   VAR_TEMP 
      tempExecute : Bool;
      tempNumberOfPoints : Int;
   END_VAR

   VAR CONSTANT 
      FB_STATE_NO_PROCESSING : DInt := 0;
      FB_STATE_ENABLE_MOVE_TO_END_POS : DInt := 3;
      FB_STATE_MOVE_TO_END_POSITION : DInt := 4;
      FB_STATE_ENABLE_RAMP_UP : DInt := 6;
      FB_STATE_RAMP_UP : DInt := 9;
      FB_STATE_WAIT_FOR_MEASUREMENT : DInt := 10;
      FB_STATE_MEASUREMENT : DInt := 11;
      FB_STATE_RAMP_DOWN : DInt := 12;
      FB_STATE_ERROR : DInt := 16;
      FB_STATE_COMMAND_ABORTED : DInt := 17;
      UNDEFINED : Byte;
      FORWARD : Byte := 16#1;
      BACKWARD : Byte := 16#2;
      FINE_RANGE : Int := 0;
      COARSE_RANGE : Int := 1;
      STATUS_MEASUREMENT_OK : Word := 16#0000;
      STATUS_MEASUREMENT_MOVE_TO_END_POS : Word := 16#0001;
      STATUS_MEASUREMENT_WAITING : Word := 16#0002;
      STATUS_MEASUREMENT_BUSY : Word := 16#0004;
      STATUS_MEASUREMENT_IS_ABORTED : Word := 16#0008;
      STATUS_MEASUREMENT_DISTANCE_TO_SMALL : Word := 16#0010;
      STATUS_MEASUREMENT_ARRAY_FORWARD_LIMITED : Word := 16#0020;
      STATUS_MEASUREMENT_ARRAY_BACKWARD_LIMITED : Word := 16#0040;
      STATUS_MEASUREMENT_ERROR : Word := 16#8000;
      STATUS_EXECUTION_FINISHED : Word := 16#0000;
      STATUS_NO_CALL : Word := 16#7000;
      STATUS_FIRST_CALL : Word := 16#7001;
      STATUS_SUBSEQUENT_CALL : Word := 16#7002;
      STATUS_WAITING_FOR_ENABLING_FORWARD : Word := 16#7003;
      STATUS_WAITING_FOR_ENABLING_BACKWARD : Word := 16#7004;
      ALARM_MEASUREMENT_IS_RUNNING : Word := 16#8201;
      ALARM_ABORT_IS_ON : Word := 16#8202;
      ALARM_UNDEFINED_STATE : Word := 16#8600;
      ALARM_VALUE_RAMP_FORWARTS : Word := 16#8005;
      ALARM_VALUE_RAMP_BACKWARDS : Word := 16#8006;
      ALARM_DIRECTION : Word := 16#8007;
      ALARM_VALUE_TRAVERSING_DISTANCE : Word := 16#8010;
      ALARM_VALUE_MAX_VELOCITY : Word := 16#8011;
      ALARM_CONFIGURATION : Word := 16#8012;
      ALARM_AXIS_ERROR_OCCURED : Word := 16#8001;
      ALARM_AXIS_DISABLED : Word := 16#800F;
   END_VAR


BEGIN
	//================================================================================
	//SIEMENS AG // (c)Copyright 2019 All Rights Reserved
	//--------------------------------------------------------------------------------
	//Library:       LSimaHydTO
	//Tested with:   S7-15xx
	//Engineering:   TIA Portal  V15
	//Restrictions:  -
	//Requirements:  S7-1500 (FW 2.5)
	//Functionality: Execute valve characteristic measurement
	//
	//--------------------------------------------------------------------------------
	//Change log table:
	//
	//Version     Date          Expert in charge    Changes applied
	//01.00    15.03.2018    APC_ERLF            First released version
	//01.22    22.04.2020    APC_ERLF              - improved: units are taken into account for the control
	//================================================================================
	#tempExecute := #execute; // Work with temporary value / create process image
	
	REGION TRIGGERING
	  IF #tempExecute AND NOT #statExecuteOld  // Check if FB is triggered
	  THEN // First call; initialize FB
	    IF #statStatus <> #STATUS_NO_CALL THEN
	      #statFBState := #FB_STATE_ERROR;
	      #statStatus := #ALARM_MEASUREMENT_IS_RUNNING;
	    ELSIF #abort THEN
	      #statFBState := #FB_STATE_ERROR;
	      #statStatus := #ALARM_ABORT_IS_ON;
	    ELSE
	      
	      #statDone := FALSE;
	      #statBusy := TRUE;
	      #statError := FALSE;
	      #statCommandAborted := FALSE;
	      #statStatus := #STATUS_FIRST_CALL;
	      
	      // reset outputs 
	      #qOutputValueStepBackward := 0.0;
	      #qOutputValueStepForward := 0.0;
	      #velocityStepBackward := 0.0;
	      #velocityStepForward := 0.0;
	      #statDirection := #UNDEFINED;
	      #statStatusMeasurement := #STATUS_MEASUREMENT_OK;
	      #statIdx := "LSIMAHYD_VCHAR_POINTS_UPPER_LIMIT" + 1;
	      
	      "LSimaHydTO_CheckPlausibilityConfigData"(forwardFineRangeStepValue => #statForwardFineRangeStepValue,
	                                               forwardCoarseRangeStepValue => #statForwardCoarseRangeStepValue,
	                                               backwardFineRangeStepValue => #statBackwardFineRangeStepValue,
	                                               backwardCoarseRangeStepValue => #statBackwardCoarseRangeStepValue,
	                                               configForwardOK => #statConfigForwardOK,
	                                               configBackwardOK => #statConfigBackwardOK,
	                                               configData := #configData);
	      
	      
	      REGION check input parameters
	        IF #axis.Internal.PositionLimits_SW.Active THEN
	          #statMaxPosition := #axis.Internal.PositionLimits_SW.MaxPosition - ABS(#configData.safetyDistance);
	          #statMinPosition := #axis.Internal.PositionLimits_SW.MinPosition + ABS(#configData.safetyDistance);
	          //check if actual position is in the limits
	        ELSE
	          #statMaxPosition := 1.0e12;
	          #statMinPosition := -1.0e12;
	          //check if actual position is in the limits
	        END_IF;
	        
	        IF #configData.forward.ramp = 0.0
	          AND #configData.forward.enableMeasurement
	        THEN
	          #statFBState := #FB_STATE_ERROR;
	          #statStatus := #ALARM_VALUE_RAMP_FORWARTS;
	        ELSIF #configData.backward.ramp = 0.0
	          AND #configData.backward.enableMeasurement
	        THEN
	          #statFBState := #FB_STATE_ERROR;
	          #statStatus := #ALARM_VALUE_RAMP_BACKWARDS;
	        ELSIF #statMaxPosition <= #statMinPosition
	          OR #configData.safetyDistance < 0.0
	        THEN
	          #statFBState := #FB_STATE_ERROR;
	          #statStatus := #ALARM_VALUE_TRAVERSING_DISTANCE;
	        ELSIF NOT (#configData.forward.enableMeasurement OR #configData.backward.enableMeasurement)
	        THEN
	          //error: no direction is enabled
	          #statFBState := #FB_STATE_ERROR;
	          #statStatus := #ALARM_DIRECTION;
	        ELSIF (#configData.forward.maxVelocity = 0.0 AND #configData.forward.enableMeasurement)
	          OR (#configData.backward.maxVelocity = 0.0 AND #configData.backward.enableMeasurement)
	        THEN
	          //error: illegal value Vmax
	          #statFBState := #FB_STATE_ERROR;
	          #statStatus := #ALARM_VALUE_MAX_VELOCITY;
	        ELSE
	          //check config forward
	          IF #statConfigForwardOK THEN
	            IF #configData.forward.fineRange.numberOfPoints > 0 THEN
	              #statRangeForward := #FINE_RANGE;
	              #statCoarseBeginForward := -1;
	            ELSE
	              #statRangeForward := #COARSE_RANGE;
	              #statCoarseBeginForward := 0;
	            END_IF;
	          END_IF;
	          //check config backward
	          IF #statConfigBackwardOK THEN
	            IF #configData.backward.fineRange.numberOfPoints > 0 THEN
	              #statRangeBackward := #FINE_RANGE;
	              #statCoarseBeginBackward := -1;
	            ELSE
	              #statRangeBackward := #COARSE_RANGE;
	              #statCoarseBeginBackward := 0;
	            END_IF;
	          END_IF;
	          IF NOT (#statConfigForwardOK OR #statConfigBackwardOK) THEN
	            //error: illegal config configuration
	            #statFBState := #FB_STATE_ERROR;
	            #statStatus := #ALARM_CONFIGURATION;
	          ELSE
	            #statError := FALSE;
	            #statStatus := #STATUS_FIRST_CALL;
	            #statStatusMeasurement := #STATUS_MEASUREMENT_OK;
	          END_IF;
	        END_IF;
	        
	        //check input parameters
	        IF #statFBState <> #FB_STATE_ERROR
	        THEN
	          //init internal variables
	          #statMeasurementForwardDone := NOT #configData.forward.enableMeasurement;
	          #statMeasurementBackwardDone := NOT #configData.backward.enableMeasurement;
	          #statActualStepForward := 0;
	          #statActualStepBackward := 0;
	          #statIdx := 0;
	          #measuredValues.forward.maxQOutput := 0.0;
	          #measuredValues.forward.maxVelocity := 0.0;
	          #measuredValues.forward.maxIndexMeasurement := -1;
	          #measuredValues.backward.maxQOutput := 0.0;
	          #measuredValues.backward.maxVelocity := 0.0;
	          #measuredValues.backward.maxIndexMeasurement := -1;
	          #statStepCounterMeasurementForwardAborted := 0;
	          #statStepCounterMeasurementBackwardAborted := 0;
	          
	        ELSE
	          //set PLCopen outputs
	          #statBusy := FALSE;
	        END_IF;
	        
	      END_REGION
	      
	    END_IF;
	  ELSIF (#statStatus = #STATUS_FIRST_CALL) THEN
	    #statStatus := #STATUS_SUBSEQUENT_CALL;
	  END_IF;
	  
	  // Edge detection 'execute' input
	  #statExecuteOld := #tempExecute;
	END_REGION TRIGGERING
	
	IF (#statStatus = #STATUS_NO_CALL) THEN // Nothing to do -> End here to reduce "system load"
	  RETURN;
	END_IF;
	
	REGION WATCHING 
	  //get actual position
	  #statActualPosition := #axis.ActualPosition;
	  //get actual Time
	  #statRetInt := RD_SYS_T(#statActualTime);
	  //init internal variables
	  
	  
	  REGION INIT_MEASUREMENT
	    IF #statStatus = #STATUS_FIRST_CALL AND NOT #statError THEN
	      #statStatusMeasurement := #statStatusMeasurement AND NOT #STATUS_MEASUREMENT_MOVE_TO_END_POS;
	      
	      IF #configData.forward.enableMeasurement AND #configData.backward.enableMeasurement THEN
	        //check start direction
	        IF (#statMaxPosition - #statActualPosition) > (#statActualPosition - #statMinPosition) THEN
	          #statDirection := #FORWARD;
	        ELSE
	          #statDirection := #BACKWARD;
	        END_IF;
	        #statFBState := #FB_STATE_ENABLE_RAMP_UP;
	      ELSE
	        IF #configData.forward.enableMeasurement THEN
	          IF #statActualPosition < #statMaxPosition - #configData.safetyDistance THEN
	            #statDirection := #FORWARD;
	            #statFBState := #FB_STATE_ENABLE_RAMP_UP;
	          ELSE
	            #statDirection := #BACKWARD;
	            #statFBState := #FB_STATE_ENABLE_MOVE_TO_END_POS;
	          END_IF;
	        ELSE
	          IF #statActualPosition > #statMinPosition + #configData.safetyDistance THEN
	            #statDirection := #BACKWARD;
	            #statFBState := #FB_STATE_ENABLE_RAMP_UP;
	          ELSE
	            #statDirection := #FORWARD;
	            #statFBState := #FB_STATE_ENABLE_MOVE_TO_END_POS;
	          END_IF;
	        END_IF;
	      END_IF;
	      //start always from min. value
	      #statQOutputForward := MAX(IN1 := #configData.forward.minQOutputValue, IN2 := #configData.offset);
	      #measuredValues.forward.minQOutput := (#configData.forward.minQOutputValue);
	      #statQOutputBackward := MAX(IN1 := ABS(#configData.backward.minQOutputValue), IN2 := ABS(#configData.offset));
	      #measuredValues.backward.minQOutput := (- #configData.backward.minQOutputValue);
	      #statEnableRamping := (#enableRampingForward AND #statDirection = #FORWARD) OR (#enableRampingBackward AND #statDirection = #BACKWARD);
	      
	    END_IF;
	  END_REGION INIT_MEASUREMENT
	  
	  
	  #statEnableRamping := (#enableRampingForward AND #statDirection = #FORWARD) OR (#enableRampingBackward AND #statDirection = #BACKWARD);
	  IF ((#axis.ErrorWord <> 0 OR NOT #axis.StatusActor.Enabled)
	    AND #statFBState <> #FB_STATE_NO_PROCESSING) OR  #statFBState = #FB_STATE_ERROR
	  THEN
	    IF #axis.ErrorWord <> 0 THEN
	      #statStatus := #ALARM_AXIS_ERROR_OCCURED;
	    ELSIF NOT #axis.StatusActor.Enabled THEN
	      #statStatus := #ALARM_AXIS_DISABLED;
	    END_IF;
	    
	    #axis.Internal.Control.DirectOutput.activate := FALSE;
	    #axis.Internal.Control.DirectOutput.jogForward := FALSE;
	    #axis.Internal.Control.DirectOutput.jogBackward := FALSE;
	    #statFBState := #FB_STATE_ERROR;
	    // stop/pause measurement
	  ELSIF (#abort AND NOT #statAbortOld)
	    OR
	    (NOT #statEnableRamping AND #statEnableRampingOld)
	  THEN
	    IF #statFBState = #FB_STATE_MOVE_TO_END_POSITION
	      OR #statFBState = #FB_STATE_RAMP_UP
	      OR #statFBState = #FB_STATE_WAIT_FOR_MEASUREMENT
	      OR #statFBState = #FB_STATE_MEASUREMENT THEN
	      #statCommandAborted := #abort;
	      #axis.Internal.Control.DirectOutput.jogForward := FALSE;
	      #axis.Internal.Control.DirectOutput.jogBackward := FALSE;
	      #statFBState := #FB_STATE_RAMP_DOWN;
	    ELSIF #abort AND #statFBState <> #FB_STATE_NO_PROCESSING
	      AND #statFBState <> #FB_STATE_ERROR
	      AND #statFBState <> #FB_STATE_COMMAND_ABORTED
	    THEN
	      #statCommandAborted := #abort;
	      #statStatusMeasurement := #STATUS_MEASUREMENT_IS_ABORTED;
	      #statFBState := #FB_STATE_COMMAND_ABORTED;
	    END_IF;
	  END_IF;
	  
	  
	  // do not use statI in a following operation
	  IF #statIdx <= "LSIMAHYD_VCHAR_POINTS_UPPER_LIMIT" THEN
	    #measuredValues.forward.qOutput[#statIdx] := 0.0;  // Q-Output value
	    #measuredValues.forward.velocity[#statIdx] := 0.0;  // velocity
	    #measuredValues.backward.qOutput[#statIdx] := 0.0;  // Q-Output value
	    #measuredValues.backward.velocity[#statIdx] := 0.0;  // velocity
	    #statIdx := #statIdx + 1;
	  END_IF;
	END_REGION
	
	REGION STATE_MACHINE
	  #statNumOfLoop := 0; // counter to avoid endless loop
	  REPEAT
	    #statFBStateOld := #statFBState;
	    #statEnableRamping := (#enableRampingForward AND #statDirection = #FORWARD) OR (#enableRampingBackward AND #statDirection = #BACKWARD);
	    
	    CASE #statFBState OF
	        
	        //do nothing
	      #FB_STATE_NO_PROCESSING:
	        
	        REGION NO_PROCESSING
	          IF NOT #statError THEN
	            #statStatus := #STATUS_NO_CALL;
	          END_IF;
	        END_REGION
	        
	        
	        //move to end position
	      #FB_STATE_ENABLE_MOVE_TO_END_POS:
	        
	        REGION WAIT_FOR_ENABLE_MOVE_TO_END_POS
	          
	          IF #statEnableRamping  THEN
	            IF #statDirection = #FORWARD THEN
	              #axis.Internal.Control.DirectOutput.commandValueRamp := #configData.forward.ramp;
	              #axis.Internal.Control.DirectOutput.commandValueForward := ABS(#configData.forward.setpointForMovement);
	              #axis.Internal.Control.DirectOutput.jogForward := TRUE;
	            ELSIF #statDirection = #BACKWARD THEN
	              #axis.Internal.Control.DirectOutput.commandValueRamp := #configData.backward.ramp;
	              #axis.Internal.Control.DirectOutput.commandValueBackward := ABS(#configData.backward.setpointForMovement);
	              #axis.Internal.Control.DirectOutput.jogBackward := TRUE;
	            END_IF;
	            #axis.Internal.Control.DirectOutput.activate := TRUE;
	            #axis.Internal.Control.DirectOutput.safetyDistance := #configData.safetyDistance;
	            #statFBState := #FB_STATE_MOVE_TO_END_POSITION;
	          ELSE
	            #statEnableRampingMeasurement := (#enableRampingForward AND #statDirection = #BACKWARD AND #statActualPosition < (#statMaxPosition - #configData.safetyDistance))
	            OR (#enableRampingBackward AND #statDirection = #FORWARD AND #statActualPosition > (#statMinPosition + #configData.safetyDistance));
	            IF #statEnableRampingMeasurement AND #continueMeasurement THEN
	              
	              IF #statDirection = #FORWARD THEN
	                #statDirection := #BACKWARD;
	              ELSIF #statDirection = #BACKWARD THEN
	                #statDirection := #BACKWARD;
	              END_IF;
	              #statFBState := #FB_STATE_ENABLE_RAMP_UP;
	            END_IF;
	          END_IF;
	          //  #statEnableRampingMeasurementOld := #statEnableRampingMeasurement;
	        END_REGION
	        
	        
	      #FB_STATE_MOVE_TO_END_POSITION:
	        
	        REGION MOVE_TO_END_POSITION
	          IF #axis.Internal.MotionData.DirectOutput.rampingDown THEN
	            IF (#statDirection = #FORWARD) THEN
	              #axis.Internal.Control.DirectOutput.jogForward := FALSE;
	            ELSE
	              #axis.Internal.Control.DirectOutput.jogBackward := FALSE;
	            END_IF;
	            
	            #statFBState := #FB_STATE_RAMP_DOWN;
	          END_IF;
	        END_REGION
	        
	        
	        //wait for enable ramp up
	      #FB_STATE_ENABLE_RAMP_UP:
	        
	        REGION WAIT_FOR_ENABLE_RAMP_UP
	          IF #statEnableRamping  THEN
	            IF #statDirection = #FORWARD THEN
	              #axis.Internal.Control.DirectOutput.commandValueRamp := #configData.forward.ramp;
	              #axis.Internal.Control.DirectOutput.commandValueForward := ABS(#statQOutputForward);
	              #axis.Internal.Control.DirectOutput.jogForward := TRUE;
	            ELSIF #statDirection = #BACKWARD THEN
	              #axis.Internal.Control.DirectOutput.commandValueRamp := #configData.backward.ramp;
	              #axis.Internal.Control.DirectOutput.commandValueBackward := ABS(#statQOutputBackward);
	              #axis.Internal.Control.DirectOutput.jogBackward := TRUE;
	            END_IF;
	            #axis.Internal.Control.DirectOutput.activate := TRUE;
	            #axis.Internal.Control.DirectOutput.safetyDistance := #configData.safetyDistance;
	            #statFBState := #FB_STATE_RAMP_UP;
	          END_IF;
	        END_REGION
	        
	        
	        //start ramp up    
	      #FB_STATE_RAMP_UP:
	        
	        REGION RAMP_UP
	          //ramp down if constant velocity can not be reached
	          IF #axis.Internal.MotionData.DirectOutput.rampingDown THEN
	            IF (#statDirection = #FORWARD) THEN
	              #statStepCounterMeasurementForwardAborted := #statStepCounterMeasurementForwardAborted + 1;
	              IF #statStepCounterMeasurementForwardAborted > #configData.numberOfRetryMeasurement THEN
	                #statMeasurementForwardDone := TRUE;
	              END_IF;
	              #axis.Internal.Control.DirectOutput.jogForward := FALSE;
	            ELSIF #statDirection = #BACKWARD THEN
	              #statStepCounterMeasurementBackwardAborted := #statStepCounterMeasurementBackwardAborted + 1;
	              IF #statStepCounterMeasurementBackwardAborted > #configData.numberOfRetryMeasurement THEN
	                #statMeasurementBackwardDone := TRUE;
	              END_IF;
	              #axis.Internal.Control.DirectOutput.jogBackward := FALSE;
	            END_IF;
	            #statFBState := #FB_STATE_RAMP_DOWN;
	          ELSE
	            //ramp up in forward direction
	            IF #statDirection = #FORWARD THEN
	              #axis.Internal.Control.DirectOutput.commandValueForward := #statQOutputForward;
	              #axis.Internal.Control.DirectOutput.commandValueRamp := #configData.forward.ramp;
	              //IF command Q-Output value is reached THEN
	              IF #axis.Internal.MotionData.DirectOutput.QOutputValue >= #statQOutputForward THEN
	                //ramp up is done
	                #statFBState := #FB_STATE_WAIT_FOR_MEASUREMENT;
	              END_IF;
	              //ramp up in backward direction
	            ELSIF #statDirection = #BACKWARD THEN
	              #axis.Internal.Control.DirectOutput.commandValueBackward := #statQOutputBackward;
	              #axis.Internal.Control.DirectOutput.commandValueRamp := #configData.backward.ramp;
	              // IF command Q-Output value is reached THEN
	              IF #axis.Internal.MotionData.DirectOutput.QOutputValue <= #statQOutputBackward * (-1.0) THEN
	                // ramp up is done
	                
	                #statFBState := #FB_STATE_WAIT_FOR_MEASUREMENT;
	              END_IF;
	            END_IF;
	            IF #statFBState = #FB_STATE_WAIT_FOR_MEASUREMENT THEN
	              
	              #instTONWaitForMeasurement(IN := FALSE,
	                                         PT := DINT_TO_TIME(ABS(#configData.waitTimeMeasurement)));
	              
	            END_IF;
	          END_IF;
	        END_REGION
	        
	        
	      #FB_STATE_WAIT_FOR_MEASUREMENT:
	        
	        REGION WAIT_FOR_MEASUREMENT
	          IF #axis.Internal.MotionData.DirectOutput.rampingDown THEN
	            IF (#statDirection = #FORWARD) THEN
	              #statStepCounterMeasurementForwardAborted := #statStepCounterMeasurementForwardAborted + 1;
	              IF #statStepCounterMeasurementForwardAborted > #configData.numberOfRetryMeasurement THEN
	                #statMeasurementForwardDone := TRUE;
	              END_IF;
	              #axis.Internal.Control.DirectOutput.jogForward := FALSE;
	            ELSIF #statDirection = #BACKWARD THEN
	              #statStepCounterMeasurementBackwardAborted := #statStepCounterMeasurementBackwardAborted + 1;
	              IF #statStepCounterMeasurementBackwardAborted > #configData.numberOfRetryMeasurement THEN
	                #statMeasurementBackwardDone := TRUE;
	              END_IF;
	              #axis.Internal.Control.DirectOutput.jogBackward := FALSE;
	            END_IF;
	            #statFBState := #FB_STATE_RAMP_DOWN;
	          ELSE
	            
	            #instTONWaitForMeasurement(IN := TRUE,
	                                       PT := DINT_TO_TIME(ABS(#configData.waitTimeMeasurement)));
	            
	            IF #instTONWaitForMeasurement.Q THEN
	              // reset start position and time for measurement
	              #statPositionMeasurementStart := #statActualPosition;
	              #statTimeMeasurementStart := #statActualTime;
	              #statFBState := #FB_STATE_MEASUREMENT;
	            END_IF;
	          END_IF;
	        END_REGION
	        
	        
	      #FB_STATE_MEASUREMENT:
	        
	        REGION MEASUREMENT
	          
	          IF #axis.Internal.MotionData.DirectOutput.rampingDown
	            OR ((#statActualTime - #statTimeMeasurementStart) >= DINT_TO_TIME(ABS(#configData.maxMeasurementTime))) THEN
	            //set measurement data
	            #statPositionMeasurementEnd := #statActualPosition;
	            #statTimeMeasurementEnd := #statActualTime;
	            IF #statDirection = #FORWARD THEN
	              #statStepCounterMeasurementForwardAborted := 0;
	              IF NOT #statMeasurementForwardDone THEN
	                #measuredValues.forward.maxIndexMeasurement := #statActualStepForward;
	                #measuredValues.forward.qOutput[#statActualStepForward] := LREAL_TO_REAL(#axis.Internal.MotionData.DirectOutput.QOutputValue);
	                IF #statActualStepForward = #statCoarseBeginForward THEN
	                  #measuredValues.forward.coarseBegin := #measuredValues.forward.qOutput[#statActualStepForward];
	                END_IF;
	                //calculate velocity to related Q-Output value
	                #measuredValues.forward.velocity[#statActualStepForward] := LREAL_TO_REAL((#statPositionMeasurementEnd - #statPositionMeasurementStart) * 1000.0
	                                                                                          * #axis.Internal.UnitsCorrection.velFactor
	                                                                                          / TIME_TO_DINT(#statTimeMeasurementEnd - #statTimeMeasurementStart));
	                //set output, velocity of last successful measured step
	                #velocityStepForward := #measuredValues.forward.velocity[#statActualStepForward];
	                //set output, Q-Output of last successful measured step
	                #qOutputValueStepForward := #statQOutputForward;
	                #measuredValues.forward.maxQOutput := #measuredValues.forward.qOutput[#statActualStepForward];
	                #measuredValues.forward.maxVelocity := MAX(IN1 := #measuredValues.forward.maxVelocity,
	                                                           IN2 := #measuredValues.forward.velocity[#statActualStepForward]);
	              END_IF;
	              IF #statQOutputForward >= ABS(#configData.forward.coarseRange.maxQOutputValue) THEN
	                #statMeasurementForwardDone := TRUE;
	              END_IF;
	              //calculate max. Q-Output value depending on max. velocity
	              IF ABS(#measuredValues.forward.maxVelocity) > ABS(#configData.forward.maxVelocity) THEN
	                IF #statActualStepForward > 0 THEN
	                  #measuredValues.forward.maxQOutput :=
	                  #measuredValues.forward.qOutput[#statActualStepForward - 1] +
	                  (#measuredValues.forward.maxQOutput - #measuredValues.forward.qOutput[#statActualStepForward - 1]) *
	                  (ABS(#configData.forward.maxVelocity) - #measuredValues.forward.velocity[#statActualStepForward - 1]) /
	                  (#measuredValues.forward.maxVelocity - #measuredValues.forward.velocity[#statActualStepForward - 1]);
	                  #measuredValues.forward.maxVelocity := ABS(#configData.forward.maxVelocity);
	                END_IF;
	                #statMeasurementForwardDone := TRUE;
	              END_IF;
	              //next increment
	              IF NOT #statMeasurementForwardDone THEN
	                IF #statRangeForward = #FINE_RANGE THEN
	                  #statQOutputForward := #statQOutputForward + ABS(#statForwardFineRangeStepValue);
	                  IF #statQOutputForward >= ABS(#configData.forward.fineRange.maxQOutputValue) THEN
	                    #statQOutputForward := ABS(#configData.forward.fineRange.maxQOutputValue);
	                    //check next increment
	                    IF #configData.forward.coarseRange.numberOfPoints > 0 THEN
	                      #statRangeForward := #COARSE_RANGE;
	                      #statCoarseBeginForward := #statActualStepForward + 1;
	                    END_IF;
	                  END_IF;
	                ELSE
	                  #statQOutputForward := MIN(IN1 := #statQOutputForward + ABS(#statForwardCoarseRangeStepValue)
	                                             , IN2 := ABS(#configData.forward.coarseRange.maxQOutputValue));
	                END_IF;
	                #tempNumberOfPoints := #measuredValues.forward.maxIndexMeasurement + #measuredValues.backward.maxIndexMeasurement + 1;
	                IF ABS(#configData.backward.minQOutputValue) > 0.0 THEN
	                  #tempNumberOfPoints := #tempNumberOfPoints + 1;
	                END_IF;
	                IF #tempNumberOfPoints > "LSIMAHYD_VCHAR_POINTS_UPPER_LIMIT" + 1
	                  OR #statActualStepForward >= "LSIMAHYD_VCHAR_POINTS_UPPER_LIMIT"
	                THEN
	                  #statStatusMeasurement := #statStatusMeasurement OR #STATUS_MEASUREMENT_ARRAY_FORWARD_LIMITED;
	                  #statMeasurementForwardDone := TRUE;
	                ELSE
	                  #statActualStepForward := #statActualStepForward + 1;
	                END_IF;
	              END_IF;
	              IF #statMeasurementForwardDone OR #axis.Internal.MotionData.DirectOutput.rampingDown THEN
	                #axis.Internal.Control.DirectOutput.jogForward := FALSE;
	                #statFBState := #FB_STATE_RAMP_DOWN;
	              ELSE
	                #axis.Internal.Control.DirectOutput.commandValueForward := #statQOutputForward;
	                #statFBState := #FB_STATE_RAMP_UP;
	              END_IF;
	            ELSIF #statDirection = #BACKWARD THEN //backward
	              #statStepCounterMeasurementBackwardAborted := 0;
	              IF NOT #statMeasurementBackwardDone THEN
	                #measuredValues.backward.maxIndexMeasurement := #statActualStepBackward;
	                #measuredValues.backward.qOutput[#statActualStepBackward] := LREAL_TO_REAL(#axis.Internal.MotionData.DirectOutput.QOutputValue);
	                IF #statActualStepBackward = #statCoarseBeginBackward THEN
	                  #measuredValues.backward.coarseBegin := #measuredValues.backward.qOutput[#statActualStepBackward];
	                END_IF;
	                //calculate velocity to related Q-Output value
	                #measuredValues.backward.velocity[#statActualStepBackward] := LREAL_TO_REAL((#statPositionMeasurementEnd - #statPositionMeasurementStart) * 1000.0
	                                                                                            * #axis.Internal.UnitsCorrection.velFactor
	                                                                                            / TIME_TO_DINT(#statTimeMeasurementEnd - #statTimeMeasurementStart));
	                //set output, velocityof last successful measured step
	                #velocityStepBackward := #measuredValues.backward.velocity[#statActualStepBackward];
	                //set output, Q-Output of last successful measured step
	                #qOutputValueStepBackward := #statQOutputBackward;
	                #measuredValues.backward.maxQOutput := #measuredValues.backward.qOutput[#statActualStepBackward];
	                #measuredValues.backward.maxVelocity := MIN(IN1 := #measuredValues.backward.maxVelocity,
	                                                            IN2 := #measuredValues.backward.velocity[#statActualStepBackward]);
	              END_IF;
	              IF #statQOutputBackward >= ABS(#configData.backward.coarseRange.maxQOutputValue) THEN
	                #statMeasurementBackwardDone := TRUE;
	              END_IF;
	              //calculate max. Q-Output value depending on max. velocity
	              IF ABS(#measuredValues.backward.maxVelocity) >= ABS(#configData.backward.maxVelocity) THEN
	                IF #statActualStepBackward > 0 THEN
	                  #measuredValues.backward.maxQOutput :=
	                  #measuredValues.backward.qOutput[#statActualStepBackward - 1] +
	                  (#measuredValues.backward.maxQOutput - #measuredValues.backward.qOutput[#statActualStepBackward - 1]) *
	                  ((-1.0) * ABS(#configData.backward.maxVelocity) - #measuredValues.backward.velocity[#statActualStepBackward - 1]) /
	                  (#measuredValues.backward.maxVelocity - #measuredValues.backward.velocity[#statActualStepBackward - 1]);
	                  #measuredValues.backward.maxVelocity := (-1.0) * ABS(#configData.backward.maxVelocity);
	                END_IF;
	                #statMeasurementBackwardDone := TRUE;
	              END_IF;
	              //next increment
	              IF NOT #statMeasurementBackwardDone THEN
	                IF #statRangeBackward = #FINE_RANGE THEN
	                  #statQOutputBackward := #statQOutputBackward + ABS(#statBackwardFineRangeStepValue);
	                  IF #statQOutputBackward >= ABS(#configData.backward.fineRange.maxQOutputValue) THEN
	                    #statQOutputBackward := ABS(#configData.backward.fineRange.maxQOutputValue);
	                    //check next increment
	                    IF #configData.backward.coarseRange.numberOfPoints > 0 THEN
	                      #statRangeBackward := #COARSE_RANGE;
	                      #statCoarseBeginBackward := #statActualStepBackward + 1;
	                    END_IF;
	                  END_IF;
	                ELSE
	                  #statQOutputBackward := MIN(IN1 := #statQOutputBackward + ABS(#statBackwardCoarseRangeStepValue)
	                                              , IN2 := ABS(#configData.backward.coarseRange.maxQOutputValue));
	                END_IF;
	                #tempNumberOfPoints := #measuredValues.forward.maxIndexMeasurement + #measuredValues.backward.maxIndexMeasurement + 1;
	                IF ABS(#configData.backward.minQOutputValue) > 0.0 THEN
	                  #tempNumberOfPoints := #tempNumberOfPoints + 1;
	                END_IF;
	                IF #tempNumberOfPoints > "LSIMAHYD_VCHAR_POINTS_UPPER_LIMIT" + 1
	                  OR #statActualStepBackward >= "LSIMAHYD_VCHAR_POINTS_UPPER_LIMIT"
	                THEN
	                  //array of measurement points backward is to small
	                  #statStatusMeasurement := #statStatusMeasurement OR #STATUS_MEASUREMENT_ARRAY_BACKWARD_LIMITED;
	                  #statMeasurementBackwardDone := TRUE;
	                ELSE
	                  #statActualStepBackward := #statActualStepBackward + 1;
	                END_IF;
	              END_IF;
	              IF #statMeasurementBackwardDone OR #axis.Internal.MotionData.DirectOutput.rampingDown THEN
	                #axis.Internal.Control.DirectOutput.jogBackward := FALSE;
	                #statFBState := #FB_STATE_RAMP_DOWN;
	              ELSE
	                #axis.Internal.Control.DirectOutput.commandValueBackward := #statQOutputBackward;
	                #statFBState := #FB_STATE_RAMP_UP;
	              END_IF;
	            END_IF;
	          END_IF;
	        END_REGION
	        
	        
	      #FB_STATE_RAMP_DOWN:
	        
	        REGION RAMP_DOWN
	          
	          IF NOT #axis.Internal.MotionData.DirectOutput.active THEN
	            //ramp up is done
	            IF #statCommandAborted THEN
	              //set PLCopen outputs
	              #statDirection := #UNDEFINED;
	              #axis.Internal.Control.DirectOutput.activate := FALSE;
	              #statFBState := #FB_STATE_COMMAND_ABORTED;
	            ELSE
	              IF #statDirection = #FORWARD THEN
	                //reset output for valve forward
	                IF NOT #statMeasurementBackwardDone THEN
	                  //measurement backward
	                  #statDirection := #BACKWARD;
	                  #statFBState := #FB_STATE_ENABLE_RAMP_UP;
	                ELSIF NOT #statMeasurementForwardDone AND #configData.backward.enableMeasurement THEN
	                  #statDirection := #BACKWARD;
	                  #statFBState := #FB_STATE_ENABLE_MOVE_TO_END_POS;
	                ELSIF #statMeasurementForwardDone THEN
	                  #statStatus := #STATUS_EXECUTION_FINISHED;
	                ELSE
	                  #statFBState := #FB_STATE_ENABLE_RAMP_UP;
	                END_IF;
	              ELSE
	                //reset output for valve Backward
	                IF NOT #statMeasurementForwardDone THEN
	                  //measurement forward
	                  #statDirection := #FORWARD;
	                  #statFBState := #FB_STATE_ENABLE_RAMP_UP;
	                ELSIF NOT #statMeasurementBackwardDone AND #configData.forward.enableMeasurement THEN
	                  #statDirection := #FORWARD;
	                  #statFBState := #FB_STATE_ENABLE_MOVE_TO_END_POS;
	                ELSIF #statMeasurementBackwardDone THEN
	                  #statStatus := #STATUS_EXECUTION_FINISHED;
	                ELSE
	                  #statFBState := #FB_STATE_ENABLE_RAMP_UP;
	                END_IF;
	              END_IF;
	            END_IF;
	            IF #statStatus = #STATUS_EXECUTION_FINISHED THEN
	              #axis.Internal.Control.DirectOutput.activate := FALSE;
	              #axis.Internal.Control.DirectOutput.jogForward := FALSE;
	              #axis.Internal.Control.DirectOutput.jogBackward := FALSE;
	              #statDirection := #UNDEFINED;
	              
	              // measurement state was not reached
	              IF #statStepCounterMeasurementForwardAborted > #configData.numberOfRetryMeasurement AND
	                #statActualStepForward > 0 THEN
	                #statActualStepForward := #statActualStepForward - 1;
	                #statStatusMeasurement := #statStatusMeasurement OR #STATUS_MEASUREMENT_DISTANCE_TO_SMALL;
	              END_IF;
	              IF #statStepCounterMeasurementBackwardAborted > #configData.numberOfRetryMeasurement AND
	                #statActualStepBackward > 0 THEN
	                #statActualStepBackward := #statActualStepBackward - 1;
	                #statStatusMeasurement := #statStatusMeasurement OR #STATUS_MEASUREMENT_DISTANCE_TO_SMALL;
	              END_IF;
	              //set PLCopen outputs
	              #statStatusMeasurement := (#statStatusMeasurement AND 16#00F0);
	            END_IF;
	          END_IF;
	        END_REGION
	        
	        
	        #FB_STATE_ERROR,
	        #FB_STATE_COMMAND_ABORTED:
	          #statDirection := #UNDEFINED;
	          #axis.Internal.Control.DirectOutput.activate := FALSE;
	          #axis.Internal.Control.DirectOutput.jogForward := FALSE;
	          #axis.Internal.Control.DirectOutput.jogBackward := FALSE;
	          
	      ELSE
	        ;
	    END_CASE;
	    
	    #statNumOfLoop := #statNumOfLoop + 1;
	  UNTIL (#statFBState = #statFBStateOld)
	    OR #statNumOfLoop >= 3
	  END_REPEAT;
	
	END_REGION STATE_MACHINE
	
	REGION OUTPUTS
	  // Write outputs
	  IF (#statStatus = #STATUS_EXECUTION_FINISHED) AND (#statDone = FALSE) THEN // Execution finished without errors
	    #statDone := TRUE;
	    #statBusy := FALSE;
	    #statError := FALSE;
	    #statCommandAborted := FALSE;
	    #statFBState := #FB_STATE_NO_PROCESSING; // Switch state machine to "no processing"
	    
	  ELSIF (#statStatus.%X15 = TRUE) AND (#statError = FALSE) THEN // Error occurred (#statStatus is 16#8000 to 16#FFFF)
	    #statDone := FALSE;
	    #statBusy := FALSE;
	    #statError := TRUE;
	    #statCommandAborted := FALSE;
	    #statFBState := #FB_STATE_NO_PROCESSING; // Switch state machine to "no processing"
	  ELSIF #statCommandAborted AND #statFBState = #FB_STATE_COMMAND_ABORTED THEN
	    #statDone := FALSE;
	    #statBusy := FALSE;
	    #statError := FALSE;
	    #statCommandAborted := TRUE;
	    #statFBState := #FB_STATE_NO_PROCESSING; // Switch state machine to "no processing"
	  ELSIF (#tempExecute = FALSE) AND ((#statDone = TRUE) OR (#statError = TRUE) OR (#statCommandAborted = TRUE))
	    AND #statFBState = #FB_STATE_NO_PROCESSING
	  THEN // Reset outputs
	    #statDone := FALSE;
	    #statBusy := FALSE;
	    #statError := FALSE;
	    #statCommandAborted := FALSE;
	    #statStatus := #STATUS_NO_CALL;
	  END_IF;
	  //move to end stop
	  #statStatusMeasurement.%X0 := (#statFBState = #FB_STATE_ENABLE_MOVE_TO_END_POS) OR (#statFBState = #FB_STATE_MOVE_TO_END_POSITION);
	  //waiting
	  #statStatusMeasurement.%X1 := (#statFBState = #FB_STATE_ENABLE_MOVE_TO_END_POS) OR (#statFBState = #FB_STATE_ENABLE_RAMP_UP);
	  //busy
	  #statStatusMeasurement.%X2 := (#statFBState = #FB_STATE_MOVE_TO_END_POSITION) OR (#statFBState = #FB_STATE_RAMP_UP) OR (#statFBState = #FB_STATE_RAMP_DOWN);
	  //aborted
	  #statStatusMeasurement.%X3 := (#statFBState = #FB_STATE_COMMAND_ABORTED);
	  // error
	  #statStatusMeasurement.%X15 := (#statFBState = #FB_STATE_ERROR);
	  
	  
	  IF #statStatus = #STATUS_NO_CALL THEN
	    #statDirection := #UNDEFINED;
	    #axis.Internal.Control.DirectOutput.activate := FALSE;
	    #axis.Internal.Control.DirectOutput.jogForward := FALSE;
	    #axis.Internal.Control.DirectOutput.jogBackward := FALSE;
	    #statStatusMeasurement := #STATUS_MEASUREMENT_OK;
	  END_IF;
	  
	  // Write static values to outputs
	  #done := #statDone;
	  #busy := #statBusy;
	  #commandAborted := #statCommandAborted;
	  #requestForward := #statDirection.%X0;
	  #requestBackward := #statDirection.%X1;
	  
	  IF #statStatus <> #STATUS_NO_CALL THEN
	    #error := #statError;
	    #status := #statStatus;
	    #statusMeasurement := #statStatusMeasurement;
	  END_IF;
	  
	END_REGION OUTPUTS  
	
	#statAbortOld := #abort;
	#statEnableRampingOld := #statEnableRamping;
	
END_FUNCTION_BLOCK

FUNCTION "LSimaHydTO_CheckPlausibilityConfigData" : Void
{ S7_Optimized_Access := 'TRUE' }
AUTHOR : APC_ERLF
FAMILY : LSimaHydTO
VERSION : 1.0
   VAR_OUTPUT 
      forwardFineRangeStepValue : Real;
      forwardCoarseRangeStepValue : Real;
      backwardFineRangeStepValue : Real;
      backwardCoarseRangeStepValue : Real;
      configForwardOK : Bool;
      configBackwardOK : Bool;
   END_VAR

   VAR_IN_OUT 
      configData : "LSimaHydTO_typeMeasurementConfig";
   END_VAR

   VAR_TEMP 
      tempForwardCalcNumOfPoints : Int;
      tempBackwardCalcNumOfPoints : Int;
   END_VAR


BEGIN
	//================================================================================
	//SIEMENS AG // (c)Copyright 2019 All Rights Reserved
	//--------------------------------------------------------------------------------
	//Library:       LSimaHydTO
	//Tested with:   S7-15xx
	//Engineering:   TIA Portal  V15
	//Restrictions:  -
	//Requirements:  S7-1500 (FW 2.5)
	//Functionality: - for internal use
	//
	//--------------------------------------------------------------------------------
	//Change log table:
	//
	//Version     Date          Expert in charge    Changes applied
	//01.00.00    15.03.2018    APC_ERLF            First released version
	//================================================================================
	
	
	//check Q-Output settings #################################################
	#configData.offset := LIMIT(MN := -100.0,  // [%]
	                                       IN := #configData.offset,
	                                       MX := +100.0  // [%]
	);
	
	//check settings forward ##################################################
	"LSimaHydTO_CheckPlausibilityConfigQOutput"(occupiedPoints := 0,
	                                            fineRangeStepValue=>#forwardFineRangeStepValue,
	                                            coarseRangeStepValue=>#forwardCoarseRangeStepValue,
	                                            calcNumOfPoints=>#tempForwardCalcNumOfPoints,
	                                            qOutputConfig := #configData.forward);
	
	#configForwardOK := #tempForwardCalcNumOfPoints > 0 AND #configData.forward.enableMeasurement;
	
	//check settings backward ##################################################
	"LSimaHydTO_CheckPlausibilityConfigQOutput"(occupiedPoints := #tempForwardCalcNumOfPoints,
	                                            fineRangeStepValue=>#backwardFineRangeStepValue,
	                                            coarseRangeStepValue=>#backwardCoarseRangeStepValue,
	                                            calcNumOfPoints=>#tempBackwardCalcNumOfPoints,
	                                            qOutputConfig := #configData.backward);
	
	#configBackwardOK := #tempBackwardCalcNumOfPoints > 0 AND #configData.backward.enableMeasurement;
	
	
END_FUNCTION

FUNCTION "LSimaHydTO_CheckPlausibilityConfigQOutput" : Void
{ S7_Optimized_Access := 'TRUE' }
AUTHOR : APC_ERLF
FAMILY : LSimaHydTO
VERSION : 1.0
   VAR_INPUT 
      occupiedPoints : DInt;
   END_VAR

   VAR_OUTPUT 
      fineRangeStepValue : Real;
      coarseRangeStepValue : Real;
      calcNumOfPoints : Int;
   END_VAR

   VAR_IN_OUT 
      qOutputConfig : "LSimaHydTO_typeMeasurementQOutput";
   END_VAR

   VAR_TEMP 
      tempOutputBegin : Real;
      tempFreePoints : DInt;
   END_VAR


BEGIN
	//================================================================================
	//SIEMENS AG // (c)Copyright 2019 All Rights Reserved
	//--------------------------------------------------------------------------------
	//Library:       LSimaHydTO
	//Tested with:   S7-15xx
	//Engineering:   TIA Portal  V15
	//Restrictions:  -
	//Requirements:  S7-1500 (FW 2.5)
	//Functionality: - for internal use
	//
	//--------------------------------------------------------------------------------
	//Change log table:
	//
	//Version     Date          Expert in charge    Changes applied
	//01.00.00    15.03.2018    APC_ERLF            First released version
	//================================================================================
	
	
	  
	IF #qOutputConfig.enableMeasurement THEN
	  #qOutputConfig.setpointForMovement := LIMIT(MN := #tempOutputBegin  // [%]
	                                              , IN := #qOutputConfig.setpointForMovement
	                                              , MX := 200.0  // [%]
	  );
	  
	  
	  //check increment settings ################################################
	  #tempFreePoints := "LSIMAHYD_VCHAR_POINTS_UPPER_LIMIT" - #occupiedPoints;
	  IF #tempFreePoints = 0 THEN
	    #qOutputConfig.fineRange.maxQOutputValue := 0.0;
	  ELSE
	    #qOutputConfig.fineRange.maxQOutputValue := LIMIT(MN := #tempOutputBegin, IN := #qOutputConfig.fineRange.maxQOutputValue, MX := 200.0);
	  END_IF;
	  IF #qOutputConfig.fineRange.maxQOutputValue = #tempOutputBegin THEN
	    #qOutputConfig.fineRange.numberOfPoints := 0;
	    #fineRangeStepValue := 0.0;
	  ELSE
	    #qOutputConfig.fineRange.numberOfPoints := DINT_TO_INT(LIMIT(MN := 1, IN := #qOutputConfig.fineRange.numberOfPoints, MX := #tempFreePoints));
	    #fineRangeStepValue := (#qOutputConfig.fineRange.maxQOutputValue - #tempOutputBegin) / #qOutputConfig.fineRange.numberOfPoints;
	  END_IF;
	  #tempFreePoints := #tempFreePoints - #qOutputConfig.fineRange.numberOfPoints;
	  IF #tempFreePoints = 0 THEN
	    #qOutputConfig.coarseRange.maxQOutputValue := #qOutputConfig.fineRange.maxQOutputValue;
	  ELSE
	    #qOutputConfig.coarseRange.maxQOutputValue := LIMIT(MN := #qOutputConfig.fineRange.maxQOutputValue, IN := #qOutputConfig.coarseRange.maxQOutputValue, MX := 200.0);
	  END_IF;
	  IF #qOutputConfig.coarseRange.maxQOutputValue = #qOutputConfig.fineRange.maxQOutputValue THEN
	    #qOutputConfig.coarseRange.numberOfPoints := 0;
	    #coarseRangeStepValue := 0.0;
	  ELSE
	    #qOutputConfig.coarseRange.numberOfPoints := DINT_TO_INT(LIMIT(MN := 1, IN := #qOutputConfig.coarseRange.numberOfPoints, MX := #tempFreePoints));
	    #coarseRangeStepValue := (#qOutputConfig.coarseRange.maxQOutputValue - #qOutputConfig.fineRange.maxQOutputValue) / #qOutputConfig.coarseRange.numberOfPoints;
	  END_IF;
	  #calcNumOfPoints := #qOutputConfig.fineRange.numberOfPoints + #qOutputConfig.coarseRange.numberOfPoints;
	ELSE
	  #calcNumOfPoints := 0;
	END_IF;
	
	
END_FUNCTION

FUNCTION_BLOCK "SimaHydTO_VCharEditor"
{ S7_Optimized_Access := 'TRUE' }
FAMILY : SimaHydTO
VERSION : 1.0
   VAR_IN_OUT 
      hmiConnection : "SimaHydTO_typeHMIConnection";
      vCharArray : Array[*] of "SimaHydTO_typeVCharArray";
   END_VAR

   VAR 
      statFirstRunDone { ExternalAccessible := 'False'; ExternalVisible := 'False'; ExternalWritable := 'False'} : Bool;
      statLoadMeasuredValuesOld { ExternalAccessible := 'False'; ExternalVisible := 'False'; ExternalWritable := 'False'} : Bool;
      statLoadVCharOld { ExternalAccessible := 'False'; ExternalVisible := 'False'; ExternalWritable := 'False'} : Bool;
      statCreateNewVCharOld { ExternalAccessible := 'False'; ExternalVisible := 'False'; ExternalWritable := 'False'} : Bool;
      statSaveVCharOld { ExternalAccessible := 'False'; ExternalVisible := 'False'; ExternalWritable := 'False'} : Bool;
      statAbortVCharOld { ExternalAccessible := 'False'; ExternalVisible := 'False'; ExternalWritable := 'False'} : Bool;
      statShowPreviousRowOld { ExternalAccessible := 'False'; ExternalVisible := 'False'; ExternalWritable := 'False'} : Bool;
      statShowNextRowOld { ExternalAccessible := 'False'; ExternalVisible := 'False'; ExternalWritable := 'False'} : Bool;
      statAddRowOld { ExternalAccessible := 'False'; ExternalVisible := 'False'; ExternalWritable := 'False'} : Bool;
      statDeleteRowOld { ExternalAccessible := 'False'; ExternalVisible := 'False'; ExternalWritable := 'False'} : Bool;
      statSortAndDisplayOld { ExternalAccessible := 'False'; ExternalVisible := 'False'; ExternalWritable := 'False'} : Bool;
      statVChar { ExternalAccessible := 'False'; ExternalVisible := 'False'; ExternalWritable := 'False'} : "LSimaHydTO_typeVCharData";
      instVCharSelectorLoad { ExternalAccessible := 'False'; ExternalVisible := 'False'; ExternalWritable := 'False'} : "SimaHydTO_HmiVCharSelector";
      instVCharSelectorSave { ExternalAccessible := 'False'; ExternalVisible := 'False'; ExternalWritable := 'False'} : "SimaHydTO_HmiVCharSelector";
      statSelectedTableIndex { ExternalAccessible := 'False'; ExternalVisible := 'False'; ExternalWritable := 'False'} : Int;
      statRetVal { ExternalAccessible := 'False'; ExternalVisible := 'False'; ExternalWritable := 'False'} : Int;
      statBusyWrite { ExternalAccessible := 'False'; ExternalVisible := 'False'; ExternalWritable := 'False'} : Bool;
      statSaveToDBL { ExternalAccessible := 'False'; ExternalVisible := 'False'; ExternalWritable := 'False'} : Bool;
      statBusyWriteArray { ExternalAccessible := 'False'; ExternalVisible := 'False'; ExternalWritable := 'False'} : Bool;
      statSaveArrayToDB { ExternalAccessible := 'False'; ExternalVisible := 'False'; ExternalWritable := 'False'} : Bool;
      statTableLowerBound { ExternalAccessible := 'False'; ExternalVisible := 'False'; ExternalWritable := 'False'} : Int := 0;
      statTableUpperBound { ExternalAccessible := 'False'; ExternalVisible := 'False'; ExternalWritable := 'False'} : Int := 19;
   END_VAR

   VAR_TEMP 
      tempVariant : Variant;
      tempErrorVariant : Int;
      tempDbAny : DB_ANY;
      tempIndex : Int;
      tempVCharIndex : Int;
      tempAddRowIndex : Int;
      tempRetValCreateVChar : DInt;
      tempTableLowerBound : DInt;
      tempTableUpperBound : DInt;
   END_VAR

   VAR CONSTANT 
      MAXIMUM_REAL : Real := 3.4E+38;
      MINIMUM_REAL : Real := -3.4E+38;
      DEFAULT_LINES : Int := 0;
   END_VAR


BEGIN
	//=============================================================================
	//SIEMENS AG
	//(c)Copyright 2016 All Rights Reserved
	//-----------------------------------------------------------------------------
	//Library:       SimaHydTO_VCharEditor
	//Tested with:   S7-1500 V2.5
	//Engineering:   TIA Portal V15
	//Restrictions:  -
	//Requirements:  S7-1500(T)
	//Functionality: Editor of the valve characteristics (New/Open/Save)
	//-----------------------------------------------------------------------------
	//Change log table:
	//Version  Date       Expert in charge Changes applied
	//01.00.00 17.07.2019 ArSc             First released version
	//=============================================================================
	
	//Array detection and initialization
	IF (#statFirstRunDone = False)
	THEN
	  //Get MIN and MAX of array indices
	  "SimaHydTO_GetRealArrayBounds"(lowerBound => #tempTableLowerBound,
	                                 upperBound => #tempTableUpperBound,
	                                 arrayOfReal := #hmiConnection.VCharEditor.Table.Velocity);
	  #statTableLowerBound := DINT_TO_INT(#tempTableLowerBound);
	  #statTableUpperBound := DINT_TO_INT(#tempTableUpperBound);
	  //Mark first run of function block
	  #statFirstRunDone := True;
	END_IF;
	
	
	  #instVCharSelectorLoad(command := #hmiConnection.VCharEditor.Command.VCharLoad,
	                         status := #hmiConnection.VCharEditor.Status.VCharLoad,
	                         vCharArray := #vCharArray);
	  
	  
	  #instVCharSelectorSave(command := #hmiConnection.VCharEditor.Command.VCharSave,
	                         status := #hmiConnection.VCharEditor.Status.VCharSave,
	                         vCharArray := #vCharArray);
	  
	  
	  //=============================================================================
	  //Reset editor data
	  //=============================================================================
	  
	  //Check, if editor is active
	  IF (#hmiConnection.VCharEditor.Status.EditorActive = False)
	  THEN
	    
	    //Reset statVChar
	(*    FOR #tempIndex := 0 TO "LSIMAHYD_VCHAR_POINTS_UPPER_LIMIT" DO
	      #statVChar.QOutput[#tempIndex] := 0.0;
	      #statVChar.Velocity[#tempIndex] := 0.0;
	      #statVChar.VelocityLimitPositive := 0.0;
	      #statVChar.VelocityLimitNegative := 0.0;
	      #statVChar.ZeroZonePositive := 0.0;
	      #statVChar.ZeroZoneNegative := 0.0;
	      #statVChar.MaxIdx := 0;
	      #statVChar.Name := WSTRING#'';
	    END_FOR;
	*)    //Reset output signal
	    #hmiConnection.VCharEditor.Status.EditorActive := False;
	    #statSaveToDBL := FALSE;
	    #statSaveArrayToDB := FALSE;
	  END_IF;
	  
	  
	  //=============================================================================
	  //Open VChar in editor
	  //=============================================================================
	  
	  IF (#hmiConnection.VCharEditor.Command.LoadVChar
	    AND NOT #statLoadVCharOld
	  //  And (#hmiConnection.VCharEditor.Status.EditorActive = False)
	    AND (#hmiConnection.VCharEditor.Status.VCharLoad.dataValid = True))
	  THEN
	    //Convert data
	    #tempVariant := DB_ANY_TO_VARIANT(in := #hmiConnection.VCharEditor.Status.VCharLoad.selectedVChar, err => #tempErrorVariant);
	    //Load VChar data
	    IF TypeOf(#tempVariant) = LSimaHydTO_typeVCharData THEN
	      //Get data from VChar
	      VariantGet(SRC := #tempVariant,
	                 DST => #statVChar);
	      //Set default name of VChar
	      #hmiConnection.VCharEditor.VCharNameToSave := #statVChar.Name;
	      //Set output signal
	      #hmiConnection.VCharEditor.Status.EditorActive := True;
	      #hmiConnection.VCharEditor.Parameter.SelectedTableIndex := #statTableLowerBound;
	      //Display VChar
	      "SimaHydTO_VCharEditorDisplayVChar"(hmiConnection := #hmiConnection,
	                                          displayVChar := #statVChar);
	      //Display Table
	      #hmiConnection.VCharEditor.Parameter.ActualTableStartIndex := #statTableLowerBound;
	      //Update displaying editor table
	      "SimaHydTO_VCharEditorUpdateTable"(hmiConnection := #hmiConnection,
	                                         updateVChar := #statVChar);
	    END_IF;
	  END_IF;
	  
	  
	  //=============================================================================
	  //Create new VChar in editor
	  //=============================================================================
	  
	  IF ((#hmiConnection.VCharEditor.Command.CreateNewVChar = True)
	    AND (#statCreateNewVCharOld = False))
	  //  And (#hmiConnection.VCharEditor.Status.EditorActive = False))
	  THEN
	    //Reset statVChar
	    FOR #tempIndex := 0 TO "LSIMAHYD_VCHAR_POINTS_UPPER_LIMIT" DO
	      #statVChar.QOutput[#tempIndex] := 0.0;
	      #statVChar.Velocity[#tempIndex] := 0.0;
	      #statVChar.VelocityLimitPositive := 0.0;
	      #statVChar.VelocityLimitNegative := 0.0;
	      #statVChar.ZeroZonePositive := 0.0;
	      #statVChar.ZeroZoneNegative := 0.0;
	      #statVChar.MaxIdx := 0;
	      #statVChar.Name := Wstring#'New VChar';
	    END_FOR;
	    //Set default name of VChar
	    #hmiConnection.VCharEditor.VCharNameToSave := #statVChar.Name;
	    //Set output signal
	    #hmiConnection.VCharEditor.Status.EditorActive := True;
	    #hmiConnection.VCharEditor.Parameter.SelectedTableIndex := #statTableLowerBound;
	    //Display VChar
	    "SimaHydTO_VCharEditorDisplayVChar"(hmiConnection := #hmiConnection,
	                                        displayVChar := #statVChar);
	    //Display Table
	    #hmiConnection.VCharEditor.Parameter.ActualTableStartIndex := #statTableLowerBound;
	    //Update displaying editor table
	    "SimaHydTO_VCharEditorUpdateTable"(hmiConnection := #hmiConnection,
	                                       updateVChar := #statVChar);
	  END_IF;
	  
	  
	  //=============================================================================
	  //Open measured values of VChar in editor
	  //=============================================================================
	  
	  IF ((#hmiConnection.VCharEditor.Command.LoadMeasuredValues = True)
	    AND (#statLoadMeasuredValuesOld = False))
	   // And (#hmiConnection.VCharEditor.Status.EditorActive = False))
	  THEN
	    //Generate VChar from measured values
	    #tempRetValCreateVChar := "LSimaHydTO_CreateVChar"(measuredValues := #hmiConnection.GetCharacteristics.MeasuredValues, vchar := #statVChar);
	    //Generation successful
	    IF (#tempRetValCreateVChar = 0)
	    THEN
	      //Set default name of VChar
	      #statVChar.Name := Wstring#'MeasuredVChar';
	      #hmiConnection.VCharEditor.VCharNameToSave := #statVChar.Name;
	      //Set output signal
	      #hmiConnection.VCharEditor.Status.EditorActive := True;
	      #hmiConnection.VCharEditor.Parameter.SelectedTableIndex := #statTableLowerBound;
	      //Display VChar
	      "SimaHydTO_VCharEditorDisplayVChar"(hmiConnection := #hmiConnection,
	                                          displayVChar := #statVChar);
	      //Display Table
	      #hmiConnection.VCharEditor.Parameter.ActualTableStartIndex := #statTableLowerBound;
	      //Update displaying editor table
	      "SimaHydTO_VCharEditorUpdateTable"(hmiConnection := #hmiConnection,
	                                         updateVChar := #statVChar);
	    ELSE
	      //Reset statVChar
	      FOR #tempIndex := 0 TO "LSIMAHYD_VCHAR_POINTS_UPPER_LIMIT" DO
	        #statVChar.QOutput[#tempIndex] := 0.0;
	        #statVChar.Velocity[#tempIndex] := 0.0;
	        #statVChar.VelocityLimitPositive := 0.0;
	        #statVChar.VelocityLimitNegative := 0.0;
	        #statVChar.ZeroZonePositive := 0.0;
	        #statVChar.ZeroZoneNegative := 0.0;
	        #statVChar.MaxIdx := 0;
	        #statVChar.Name := Wstring#'';
	      END_FOR;
	      //Reset output signal
	      #hmiConnection.VCharEditor.Status.EditorActive := False;
	    END_IF;
	  END_IF;
	  
	  
	  //=============================================================================
	  //Save VChar
	  //=============================================================================
	  
	  IF ((#hmiConnection.VCharEditor.Command.SaveVChar = True)
	    AND (#statSaveVCharOld = False)
	    AND (#hmiConnection.VCharEditor.Status.EditorActive = True)
	    AND (#hmiConnection.VCharEditor.Status.VCharSave.dataValid))
	  THEN
	    //Convert data
	    #tempVariant := DB_ANY_TO_VARIANT(in := #hmiConnection.VCharEditor.Status.VCharSave.selectedVChar, err => #tempErrorVariant);
	    //Write back VChar data
	    IF TypeOf(#tempVariant) = LSimaHydTO_typeVCharData THEN
	      //Set name of VChar
	      #statVChar.Name := #hmiConnection.VCharEditor.VCharNameToSave;
	      //Write data from VChar
	      //Start sorting editor table
	      "SimaHydTO_VCharEditorSortTable"(hmiConnection := #hmiConnection,
	                                       sortVChar := #statVChar);
	      //Update displaying editor table
	      "SimaHydTO_VCharEditorUpdateTable"(hmiConnection := #hmiConnection,
	                                         updateVChar := #statVChar);
	      //Display VChar
	      "SimaHydTO_VCharEditorDisplayVChar"(hmiConnection := #hmiConnection,
	                                          displayVChar := #statVChar);
	      
	      
	      VariantPut(SRC := #statVChar,
	                 DST := #tempVariant);
	      #hmiConnection.VCharEditor.Status.VCharSave.selectedVCharName := #statVChar.Name;
	      IF #hmiConnection.VCharEditor.Status.VCharLoad.selectedVChar = #hmiConnection.VCharEditor.Status.VCharSave.selectedVChar
	      THEN
	        #hmiConnection.VCharEditor.Status.VCharLoad.selectedVCharName := #statVChar.Name;
	      END_IF;
	      
	      
	      #statSaveToDBL := TRUE;
	      #statSaveArrayToDB := TRUE;
	      //Convert data
	     // #hmiConnection.VCharEditor.Status.VCharSave.selectedVChar := VARIANT_TO_DB_ANY(in := #tempVariant, err => #tempErrorVariant);
	      //Reset VChar data of HMI
	      FOR #tempIndex := #statTableLowerBound TO #statTableUpperBound DO
	        #hmiConnection.VCharEditor.Table.Appearance[#tempIndex] := 0;
	        #hmiConnection.VCharEditor.Table.Index[#tempIndex] := 0;
	        #hmiConnection.VCharEditor.Table.Velocity[#tempIndex] := 0.0;
	        #hmiConnection.VCharEditor.Table.QOutput[#tempIndex] := 0.0;
	      END_FOR;
	      //Reset name of VChar
	      #hmiConnection.VCharEditor.VCharNameToSave := Wstring#'';
	      //Reset output signal
	      #hmiConnection.VCharEditor.Status.EditorActive := False;
	      //Display VChar
	      "SimaHydTO_VCharEditorDisplayVChar"(hmiConnection := #hmiConnection,
	                                          displayVChar := #statVChar);
	      //Display Table
	      #hmiConnection.VCharEditor.Parameter.ActualTableStartIndex := #statTableLowerBound;
	    END_IF;
	  END_IF;
	  // write DBL
	  IF #statSaveToDBL THEN
	    #tempVariant := DB_ANY_TO_VARIANT(in := #hmiConnection.VCharEditor.Status.VCharSave.selectedVChar, err => #tempErrorVariant);
	    #statRetVal := WRIT_DBL(REQ := TRUE, SRCBLK := #tempVariant, BUSY => #statBusyWrite, DSTBLK => #tempVariant);
	    IF NOT #statBusyWrite THEN
	      #statSaveToDBL := FALSE;
	    END_IF;
	  END_IF;
	  
	  // save array element
	  IF #statSaveArrayToDB THEN
	    #statRetVal := WRIT_DBL(REQ := TRUE,
	                            SRCBLK := #vCharArray[#hmiConnection.VCharEditor.Status.VCharSave.actualVCharIndex].VChar_DB,
	                            BUSY => #statBusyWriteArray,
	                            DSTBLK => #vCharArray[#hmiConnection.VCharEditor.Status.VCharSave.actualVCharIndex].VChar_DB);
	    IF NOT #statBusyWriteArray THEN
	      #statSaveArrayToDB := FALSE;
	    END_IF;
	  END_IF;
	  
	  
	  
	  //=============================================================================
	  //Abort editor (Discard VChar data)
	  //=============================================================================
	  
	  IF ((#hmiConnection.VCharEditor.Command.AbortEditor = True)
	    AND (#statAbortVCharOld = False)
	    AND (#hmiConnection.VCharEditor.Status.EditorActive = True))
	  THEN
	    //Reset VChar data of HMI
	    FOR #tempIndex := #statTableLowerBound TO #statTableUpperBound DO
	      #hmiConnection.VCharEditor.Table.Appearance[#tempIndex] := 0;
	      #hmiConnection.VCharEditor.Table.Index[#tempIndex] := 0;
	      #hmiConnection.VCharEditor.Table.Velocity[#tempIndex] := 0.0;
	      #hmiConnection.VCharEditor.Table.QOutput[#tempIndex] := 0.0;
	    END_FOR;
	    //Reset name of VChar
	    #hmiConnection.VCharEditor.VCharNameToSave := Wstring#'';
	    //Reset start index
	    #hmiConnection.VCharEditor.Parameter.ActualTableStartIndex := #statTableLowerBound;
	    //Display VChar
	    "SimaHydTO_VCharEditorDisplayVChar"(hmiConnection := #hmiConnection,
	                                        displayVChar := #statVChar);
	    // //Display Table
	    // #statUpdateTable := True;
	    //Reset output signal
	    #hmiConnection.VCharEditor.Status.EditorActive := False;
	  END_IF;
	  
	  
	  
	  
	  
	  //=============================================================================
	  //Editor function: Show previous/next row (table data)
	  //=============================================================================
	  
	  //Load previous table data
	  IF ((#hmiConnection.VCharEditor.Command.ShowPreviousRow = True)
	    AND (#statShowPreviousRowOld = False)
	    AND (#hmiConnection.VCharEditor.Status.EditorActive = True))
	  THEN
	    IF ((#hmiConnection.VCharEditor.Parameter.ActualTableStartIndex - #statTableUpperBound - 1) >= 0)
	    THEN
	      //Save actual table from HMI to VChar data
	      FOR #tempIndex := #statTableLowerBound TO #statTableUpperBound DO
	        #tempVCharIndex := #tempIndex + #hmiConnection.VCharEditor.Parameter.ActualTableStartIndex;
	        IF ((#tempVCharIndex <= #statVChar.MaxIdx)
	          AND (#hmiConnection.VCharEditor.Table.Appearance[#tempIndex]  > 0))
	        THEN
	          #statVChar.Velocity[#tempVCharIndex] := #hmiConnection.VCharEditor.Table.Velocity[#tempIndex];
	          #statVChar.QOutput[#tempVCharIndex] := #hmiConnection.VCharEditor.Table.QOutput[#tempIndex];
	        END_IF;
	      END_FOR;
	      //Set new start index
	      #hmiConnection.VCharEditor.Parameter.ActualTableStartIndex := #hmiConnection.VCharEditor.Parameter.ActualTableStartIndex - #statTableUpperBound - 1;
	      //Update displaying editor table
	      "SimaHydTO_VCharEditorUpdateTable"(hmiConnection := #hmiConnection,
	                                         updateVChar := #statVChar);
	    END_IF;
	  END_IF;
	  
	  //Load next table data
	  IF ((#hmiConnection.VCharEditor.Command.ShowNextRow = True)
	    AND (#statShowNextRowOld = False)
	    AND (#hmiConnection.VCharEditor.Status.EditorActive = True))
	  THEN
	    IF ((#hmiConnection.VCharEditor.Parameter.ActualTableStartIndex + #statTableUpperBound + 1) <= #statVChar.MaxIdx)
	    THEN
	      //Save actual table from HMI to VChar data
	      FOR #tempIndex := #statTableLowerBound TO #statTableUpperBound DO
	        #tempVCharIndex := #tempIndex + #hmiConnection.VCharEditor.Parameter.ActualTableStartIndex;
	        IF ((#tempVCharIndex <= #statVChar.MaxIdx)
	          AND (#hmiConnection.VCharEditor.Table.Appearance[#tempIndex]  > 0))
	        THEN
	          #statVChar.Velocity[#tempVCharIndex] := #hmiConnection.VCharEditor.Table.Velocity[#tempIndex];
	          #statVChar.QOutput[#tempVCharIndex] := #hmiConnection.VCharEditor.Table.QOutput[#tempIndex];
	        END_IF;
	      END_FOR;
	      //Set new start index
	      #hmiConnection.VCharEditor.Parameter.ActualTableStartIndex := #hmiConnection.VCharEditor.Parameter.ActualTableStartIndex + #statTableUpperBound + 1;
	      //Update displaying editor table
	      "SimaHydTO_VCharEditorUpdateTable"(hmiConnection := #hmiConnection,
	                                         updateVChar := #statVChar);
	    END_IF;
	  END_IF;
	  
	  
	  
	  
	  //=============================================================================
	  //Editor function: Add row to table data
	  //=============================================================================
	  
	  IF ((#hmiConnection.VCharEditor.Command.AddRow = True)
	    AND (#statAddRowOld = False)
	    AND (#hmiConnection.VCharEditor.Status.EditorActive = True))
	  THEN
	    //Check table index
	    IF (#statVChar.MaxIdx < "LSIMAHYD_VCHAR_POINTS_UPPER_LIMIT")
	    THEN
	      //Reset error bit
	      #hmiConnection.VCharEditor.Status.Error := False;
	      //Save actual table from HMI to VChar data
	      FOR #tempIndex := #statTableLowerBound TO #statTableUpperBound DO
	        #tempVCharIndex := #tempIndex + #hmiConnection.VCharEditor.Parameter.ActualTableStartIndex;
	        IF ((#tempVCharIndex <= #statVChar.MaxIdx)
	          AND (#hmiConnection.VCharEditor.Table.Appearance[#tempIndex]  > 0))
	        THEN
	          #statVChar.Velocity[#tempVCharIndex] := #hmiConnection.VCharEditor.Table.Velocity[#tempIndex];
	          #statVChar.QOutput[#tempVCharIndex] := #hmiConnection.VCharEditor.Table.QOutput[#tempIndex];
	        END_IF;
	      END_FOR;
	      //Get row index to add row
	      #tempAddRowIndex := #hmiConnection.VCharEditor.Parameter.ActualTableStartIndex + #hmiConnection.VCharEditor.Parameter.SelectedTableIndex;
	      FOR #tempIndex := #statVChar.MaxIdx TO #tempAddRowIndex BY (-1)
	      DO
	        #statVChar.Velocity[#tempIndex + 1] := #statVChar.Velocity[#tempIndex];
	        #statVChar.QOutput[#tempIndex + 1] := #statVChar.QOutput[#tempIndex];
	      END_FOR;
	      //Reset added row
	      #statVChar.Velocity[#tempAddRowIndex] := 0.0;
	      #statVChar.QOutput[#tempAddRowIndex] := 0.0;
	      //Add row to MaxIdx
	      #statVChar.MaxIdx := #statVChar.MaxIdx + 1;
	      //Select new row
	     // #hmiConnection.VCharEditor.Parameter.SelectedTableIndex := #hmiConnection.VCharEditor.Parameter.SelectedTableIndex;
	      IF (#hmiConnection.VCharEditor.Parameter.SelectedTableIndex > #statTableUpperBound)
	      THEN
	        #hmiConnection.VCharEditor.Parameter.SelectedTableIndex := #statTableUpperBound;
	      END_IF;
	    ELSE
	      //Set error bit
	      #hmiConnection.VCharEditor.Status.Error := True;
	    END_IF;
	    //Update displaying editor table
	    "SimaHydTO_VCharEditorUpdateTable"(hmiConnection := #hmiConnection,
	                                       updateVChar := #statVChar);
	  END_IF;
	  
	  
	  //=============================================================================
	  //Editor function: Delete row from table data
	  //=============================================================================
	  
	  IF ((#hmiConnection.VCharEditor.Command.DeleteRow = True)
	    AND (#statDeleteRowOld = False)
	    AND (#hmiConnection.VCharEditor.Status.EditorActive = True))
	  THEN
	    //Check table index
	    IF (0 < #statVChar.MaxIdx)
	    THEN
	      //Reset error bit
	      #hmiConnection.VCharEditor.Status.Error := False;
	      //Save actual table from HMI to VChar data
	      FOR #tempIndex := #statTableLowerBound TO #statTableUpperBound DO
	        #tempVCharIndex := #tempIndex + #hmiConnection.VCharEditor.Parameter.ActualTableStartIndex;
	        IF ((#tempVCharIndex <= #statVChar.MaxIdx)
	          AND (#hmiConnection.VCharEditor.Table.Appearance[#tempIndex]  > 0))
	        THEN
	          #statVChar.Velocity[#tempVCharIndex] := #hmiConnection.VCharEditor.Table.Velocity[#tempIndex];
	          #statVChar.QOutput[#tempVCharIndex] := #hmiConnection.VCharEditor.Table.QOutput[#tempIndex];
	        END_IF;
	      END_FOR;
	      //Get row index to delete row
	      #tempAddRowIndex := #hmiConnection.VCharEditor.Parameter.ActualTableStartIndex + #hmiConnection.VCharEditor.Parameter.SelectedTableIndex;
	      FOR #tempIndex := #tempAddRowIndex TO (#statVChar.MaxIdx - 1) BY (+1)
	      DO
	        #statVChar.Velocity[#tempIndex] := #statVChar.Velocity[#tempIndex + 1];
	        #statVChar.QOutput[#tempIndex] := #statVChar.QOutput[#tempIndex + 1];
	      END_FOR;
	      //Reset last row
	      #statVChar.Velocity[#statVChar.MaxIdx] := 0.0;
	      #statVChar.QOutput[#statVChar.MaxIdx] := 0.0;
	      //Add row to MaxIdx
	      #statVChar.MaxIdx := #statVChar.MaxIdx - 1;
	      //Select new row
	      #hmiConnection.VCharEditor.Parameter.SelectedTableIndex := #hmiConnection.VCharEditor.Parameter.SelectedTableIndex - 1;
	      IF (#hmiConnection.VCharEditor.Parameter.SelectedTableIndex < #statTableLowerBound)
	      THEN
	        #hmiConnection.VCharEditor.Parameter.SelectedTableIndex := #statTableLowerBound;
	      END_IF;
	    ELSE
	      //Set error bit
	      #hmiConnection.VCharEditor.Status.Error := True;
	    END_IF;
	    //Update displaying editor table
	    "SimaHydTO_VCharEditorUpdateTable"(hmiConnection := #hmiConnection,
	                                       updateVChar := #statVChar);
	  END_IF;
	  
	  //=============================================================================
	  //Editor function: Sort and display table data (Update table and graphics)
	  //=============================================================================
	  
	  IF ((#hmiConnection.VCharEditor.Command.SortAndDisplay = True)
	    AND (#statSortAndDisplayOld = False))
	  THEN
	    //Set output signal
	    #hmiConnection.VCharEditor.Status.Busy := True;
	    //Start sorting editor table
	    "SimaHydTO_VCharEditorSortTable"(hmiConnection := #hmiConnection,
	                                     sortVChar := #statVChar);
	    //Update displaying editor table
	    "SimaHydTO_VCharEditorUpdateTable"(hmiConnection := #hmiConnection,
	                                       updateVChar := #statVChar);
	    //Display VChar
	    "SimaHydTO_VCharEditorDisplayVChar"(hmiConnection := #hmiConnection,
	                                        displayVChar := #statVChar);
	    //Reset output signal
	    #hmiConnection.VCharEditor.Status.Busy := False;
	  END_IF;
	 (* 
	  IF #statSelectedTableIndex <> #hmiConnection.VCharEditor.Parameter.SelectedTableIndex THEN
	    FOR #tempIndex := #TABLE_MIN_INDEX TO #TABLE_MAX_INDEX DO
	      IF #hmiConnection.VCharEditor.Table.Appearance[#tempIndex] > 0 THEN
	        IF #tempIndex = #hmiConnection.VCharEditor.Parameter.SelectedTableIndex THEN
	          #hmiConnection.VCharEditor.Table.Appearance[#tempIndex] := 2;
	        ELSE
	          #hmiConnection.VCharEditor.Table.Appearance[#tempIndex] := 1;
	        END_IF;
	      END_IF;
	    END_FOR;
	  END_IF;
	  *)
	  //=============================================================================
	  //Global editor functions
	  //=============================================================================
	  
	  //Generate output data
	  IF (#hmiConnection.VCharEditor.Status.EditorActive = True)
	  THEN
	    #hmiConnection.VCharEditor.Parameter.MaximumNumberOfLines := "LSIMAHYD_VCHAR_POINTS_UPPER_LIMIT";
	    #hmiConnection.VCharEditor.Parameter.NumberOfUsedLines := #statVChar.MaxIdx;
	    #hmiConnection.VCharEditor.Parameter.NumberOfUsableLines := #hmiConnection.VCharEditor.Parameter.MaximumNumberOfLines - #hmiConnection.VCharEditor.Parameter.NumberOfUsedLines;
	  ELSE
	    #hmiConnection.VCharEditor.Parameter.MaximumNumberOfLines := #DEFAULT_LINES;
	    #hmiConnection.VCharEditor.Parameter.NumberOfUsedLines := #DEFAULT_LINES;
	    #hmiConnection.VCharEditor.Parameter.NumberOfUsableLines := #DEFAULT_LINES;
	  END_IF;
	  
	  
	  //Save data from last cycle
	  #statLoadMeasuredValuesOld := #hmiConnection.VCharEditor.Command.LoadMeasuredValues;
	  #statLoadVCharOld := #hmiConnection.VCharEditor.Command.LoadVChar;
	  #statCreateNewVCharOld := #hmiConnection.VCharEditor.Command.CreateNewVChar;
	  #statSaveVCharOld := #hmiConnection.VCharEditor.Command.SaveVChar;
	  #statAbortVCharOld := #hmiConnection.VCharEditor.Command.AbortEditor;
	  #statShowPreviousRowOld := #hmiConnection.VCharEditor.Command.ShowPreviousRow;
	  #statShowNextRowOld := #hmiConnection.VCharEditor.Command.ShowNextRow;
	  #statAddRowOld := #hmiConnection.VCharEditor.Command.AddRow;
	  #statDeleteRowOld := #hmiConnection.VCharEditor.Command.DeleteRow;
	  #statSortAndDisplayOld := #hmiConnection.VCharEditor.Command.SortAndDisplay;
	  #statSelectedTableIndex := #hmiConnection.VCharEditor.Parameter.SelectedTableIndex;
	
	
	
END_FUNCTION_BLOCK

FUNCTION "SimaHydTO_GetRealArrayBounds" : Void
{ S7_Optimized_Access := 'TRUE' }
FAMILY : SimaHydTO
VERSION : 1.0
   VAR_OUTPUT 
      lowerBound : DInt;
      upperBound : DInt;
   END_VAR

   VAR_IN_OUT 
      arrayOfReal : Array[*] of Real;
   END_VAR


BEGIN
	//=============================================================================
	//SIEMENS AG
	//(c)Copyright 2016 All Rights Reserved
	//-----------------------------------------------------------------------------
	//Library:       SimaHydTO_VCharEditorDisplayVChar
	//Tested with:   S7-1500 V2.5
	//Engineering:   TIA Portal V15
	//Restrictions:  -
	//Requirements:  S7-1500(T)
	//Functionality: Check array dimensions
	//-----------------------------------------------------------------------------
	//Change log table:
	//Version  Date       Expert in charge Changes applied
	//01.00.00 25.10.2019 ArSc             First released version
	//=============================================================================
	
	
	#lowerBound := (LOWER_BOUND(ARR := #arrayOfReal, DIM := 1));
	#upperBound := (UPPER_BOUND(ARR := #arrayOfReal, DIM := 1));
	
END_FUNCTION

FUNCTION "SimaHydTO_VCharEditorDisplayVChar" : Void
{ S7_Optimized_Access := 'TRUE' }
FAMILY : SimaHydTO
VERSION : 1.0
   VAR_IN_OUT 
      hmiConnection : "SimaHydTO_typeHMIConnection";
      displayVChar : "LSimaHydTO_typeVCharData";
   END_VAR

   VAR_TEMP 
      tempIndex : Int;
      tempIndex2 : Int;
      tempVCharIndex : Int;
      tempDeltaQ : Real;
      tempActualQ : Real;
   END_VAR

   VAR CONSTANT 
      MAXIMUM_REAL : Real := 3.4E+38;
      MINIMUM_REAL : Real := -3.4E+38;
      INDEX_DATATABLE_START : Int := 1;
      INDEX_DATATABLE_ZERO : Int := 100;
      INDEX_DATATABLE_END : Int := 200;
      DEFAULT_INDEX : Int := 0;
      DEFAULT_VELOCITY : Real := 0.0;
      DEFAULT_QOUTPUT : Real := 0.0;
   END_VAR


BEGIN
	//=============================================================================
	//SIEMENS AG
	//(c)Copyright 2016 All Rights Reserved
	//-----------------------------------------------------------------------------
	//Library:       SimaHydTO_VCharEditorDisplayVChar
	//Tested with:   S7-1500 V2.5
	//Engineering:   TIA Portal V15
	//Restrictions:  -
	//Requirements:  S7-1500(T)
	//Functionality: Displaying VChar on HMI
	//-----------------------------------------------------------------------------
	//Change log table:
	//Version  Date       Expert in charge Changes applied
	//01.00.00 17.07.2019 ArSc             First released version
	//=============================================================================
	
	
	//Preset data
	#hmiConnection.HmiData.VChar.HMI_VChar_MaxQOutput := #MINIMUM_REAL;
	#hmiConnection.HmiData.VChar.HMI_VChar_MinQOutput := #MAXIMUM_REAL;
	#hmiConnection.HmiData.VChar.HMI_VCHar_MaxVelocity := #MINIMUM_REAL;
	#hmiConnection.HmiData.VChar.HMI_VChar_MinVelocity := #MAXIMUM_REAL;
	
	//Get VChar data (min/max)
	FOR #tempIndex := 0 TO #displayVChar.MaxIdx DO
	  //Check QOutput
	  IF (#displayVChar.QOutput[#tempIndex] > #hmiConnection.HmiData.VChar.HMI_VChar_MaxQOutput)
	  THEN
	    #hmiConnection.HmiData.VChar.HMI_VChar_MaxQOutput := #displayVChar.QOutput[#tempIndex];
	  END_IF;
	  IF (#displayVChar.QOutput[#tempIndex] < #hmiConnection.HmiData.VChar.HMI_VChar_MinQOutput)
	  THEN
	    #hmiConnection.HmiData.VChar.HMI_VChar_MinQOutput := #displayVChar.QOutput[#tempIndex];
	  END_IF;
	  //Check velocity
	  IF (#displayVChar.Velocity[#tempIndex] > #hmiConnection.HmiData.VChar.HMI_VCHar_MaxVelocity)
	  THEN
	    #hmiConnection.HmiData.VChar.HMI_VCHar_MaxVelocity := #displayVChar.Velocity[#tempIndex];
	  END_IF;
	  IF (#displayVChar.Velocity[#tempIndex] < #hmiConnection.HmiData.VChar.HMI_VChar_MinVelocity)
	  THEN
	    #hmiConnection.HmiData.VChar.HMI_VChar_MinVelocity := #displayVChar.Velocity[#tempIndex];
	  END_IF;
	END_FOR;
	
	//Calculate DeltaQ for HMI display
	#tempDeltaQ := (#hmiConnection.HmiData.VChar.HMI_VChar_MaxQOutput - #hmiConnection.HmiData.VChar.HMI_VChar_MinQOutput) / (#INDEX_DATATABLE_END - 1);
	//Calculate display points for HMI
	FOR #tempIndex := #INDEX_DATATABLE_START TO #INDEX_DATATABLE_END DO
	  //Do calculation
	  #tempActualQ := #hmiConnection.HmiData.VChar.HMI_VChar_MinQOutput + (#tempDeltaQ * (#tempIndex - #INDEX_DATATABLE_START));
	  IF (#tempIndex = #INDEX_DATATABLE_START)
	  THEN
	    #hmiConnection.HmiData.VChar.HMI_VChar[#tempIndex] := #displayVChar.Velocity[0];
	  ELSE
	    //Search for VChar segment
	    #tempIndex2 := 0;
	    WHILE ((#tempIndex2 < #displayVChar.MaxIdx)
	      AND NOT ((#displayVChar.QOutput[#tempIndex2] <= #tempActualQ)
	      AND (#tempActualQ <= #displayVChar.QOutput[#tempIndex2 + 1])))
	    DO
	      #tempIndex2 := #tempIndex2 + 1;
	    END_WHILE;
	    //Calculate interpolated value
	    IF (#tempActualQ <= #hmiConnection.HmiData.VChar.HMI_VChar_MaxQOutput)
	    THEN
	      //Chack calculation, if possible
	      IF ((#displayVChar.QOutput[#tempIndex2 + 1] - #displayVChar.QOutput[#tempIndex2]) <> 0.0)
	      THEN
	        //Calcualte interpolation point
	        #hmiConnection.HmiData.VChar.HMI_VChar[#tempIndex] :=
	        #displayVChar.Velocity[#tempIndex2] +
	        ((#displayVChar.Velocity[#tempIndex2 + 1] - #displayVChar.Velocity[#tempIndex2]) /
	        (#displayVChar.QOutput[#tempIndex2 + 1] - #displayVChar.QOutput[#tempIndex2])) *
	        (#tempActualQ - #displayVChar.QOutput[#tempIndex2]);
	      ELSE
	        //Take last value
	        #hmiConnection.HmiData.VChar.HMI_VChar[#tempIndex] := #hmiConnection.HmiData.VChar.HMI_VChar[#tempIndex - 1];
	      END_IF;
	    ELSE
	      //Take maximum value
	      #hmiConnection.HmiData.VChar.HMI_VChar[#tempIndex] := #hmiConnection.HmiData.VChar.HMI_VCHar_MaxVelocity;
	    END_IF;
	  END_IF;
	END_FOR;
	
	//Display VChar on trend view
	#hmiConnection.HmiData.VChar.HMI_VChar_TrendTransfer := W#16#8001;
	
END_FUNCTION

FUNCTION "SimaHydTO_VCharEditorUpdateTable" : Void
{ S7_Optimized_Access := 'TRUE' }
FAMILY : SimaHydTO
VERSION : 1.0
   VAR_IN_OUT 
      hmiConnection : "SimaHydTO_typeHMIConnection";
      updateVChar : "LSimaHydTO_typeVCharData";
   END_VAR

   VAR_TEMP 
      tempIndex : Int;
      tempVCharIndex : Int;
      tempTableLowerBound : DInt;
      tempTableUpperBound : DInt;
   END_VAR

   VAR CONSTANT 
      DEFAULT_INDEX : Int := 0;
      DEFAULT_VELOCITY : Real := 0.0;
      DEFAULT_QOUTPUT : Real := 0.0;
   END_VAR


BEGIN
	//=============================================================================
	//SIEMENS AG
	//(c)Copyright 2016 All Rights Reserved
	//-----------------------------------------------------------------------------
	//Library:       SimaHydTO_VCharEditorUpdateTable
	//Tested with:   S7-1500 V2.5
	//Engineering:   TIA Portal V15
	//Restrictions:  -
	//Requirements:  S7-1500(T)
	//Functionality: Update editor table displayed on HMI
	//-----------------------------------------------------------------------------
	//Change log table:
	//Version  Date       Expert in charge Changes applied
	//01.00.00 17.07.2019 ArSc             First released version
	//=============================================================================
	
	"SimaHydTO_GetRealArrayBounds"(lowerBound => #tempTableLowerBound,
	                               upperBound => #tempTableUpperBound,
	                               arrayOfReal := #hmiConnection.VCharEditor.Table.Velocity);
	
	//Refill editor table
	FOR #tempIndex := #tempTableLowerBound TO #tempTableUpperBound DO
	  #tempVCharIndex := #tempIndex + #hmiConnection.VCharEditor.Parameter.ActualTableStartIndex;
	  IF (#tempVCharIndex <= #updateVChar.MaxIdx)
	  THEN
	    (*
	    IF #tempVCharIndex = #hmiConnection.VCharEditor.Parameter.SelectedTableIndex THEN
	      #hmiConnection.VCharEditor.Table.Appearance[#tempIndex] := 2;
	    ELSE
	      #hmiConnection.VCharEditor.Table.Appearance[#tempIndex] := 1;
	    END_IF;
	    *)
	    #hmiConnection.VCharEditor.Table.Appearance[#tempIndex] := 1; // only visibility yet
	    #hmiConnection.VCharEditor.Table.Index[#tempIndex] := #tempVCharIndex;
	    #hmiConnection.VCharEditor.Table.Velocity[#tempIndex] := #updateVChar.Velocity[#tempVCharIndex];
	    #hmiConnection.VCharEditor.Table.QOutput[#tempIndex] := #updateVChar.QOutput[#tempVCharIndex];
	  ELSE
	    #hmiConnection.VCharEditor.Table.Appearance[#tempIndex] := 0;
	    #hmiConnection.VCharEditor.Table.Index[#tempIndex] := #DEFAULT_INDEX;
	    #hmiConnection.VCharEditor.Table.Velocity[#tempIndex] := #DEFAULT_VELOCITY;
	    #hmiConnection.VCharEditor.Table.QOutput[#tempIndex] := #DEFAULT_QOUTPUT;
	  END_IF;
	END_FOR;
	
	#hmiConnection.VCharEditor.Table.VelocityLimitNegative := #updateVChar.VelocityLimitNegative;
	#hmiConnection.VCharEditor.Table.VelocityLimitPositive := #updateVChar.VelocityLimitPositive;
	#hmiConnection.VCharEditor.Table.ZeroZoneNegative := #updateVChar.ZeroZoneNegative;
	#hmiConnection.VCharEditor.Table.ZeroZonePositive := #updateVChar.ZeroZonePositive;
	
	
	
	
	
	
	
END_FUNCTION

FUNCTION "LSimaHydTO_CreateVChar" : DInt
{ S7_Optimized_Access := 'TRUE' }
AUTHOR : APC_ERLF
FAMILY : LSimaHydTO
VERSION : 1.0
   VAR_IN_OUT 
      measuredValues : "LSimaHydTO_typeMeasuredValues";
      vchar : "LSimaHydTO_typeVCharData";
   END_VAR

   VAR_TEMP 
      tempIdx : Int;
      tmpNumOfPoints : Int;
   END_VAR


BEGIN
	//================================================================================
	//SIEMENS AG // (c)Copyright 2019 All Rights Reserved
	//--------------------------------------------------------------------------------
	//Library:       LSimaHydTO
	//Tested with:   S7-15xx
	//Engineering:   TIA Portal  V15
	//Restrictions:  -
	//Requirements:  S7-1500 (FW 2.5)
	//Functionality: Create valve characteristic from measured data
	//
	//--------------------------------------------------------------------------------
	//Change log table:
	//
	//Version     Date          Expert in charge    Changes applied
	//01.00.00    15.03.2018    APC_ERLF            First released version
	//================================================================================
	
	
	#tmpNumOfPoints := #measuredValues.forward.maxIndexMeasurement + #measuredValues.backward.maxIndexMeasurement + 1;
	IF ABS(#measuredValues.backward.minQOutput) > 0.0 THEN
	  #tmpNumOfPoints := #tmpNumOfPoints + 1;
	END_IF;
	IF #tmpNumOfPoints  > "LSIMAHYD_VCHAR_POINTS_UPPER_LIMIT" + 1 THEN
	  #LSimaHydTO_CreateVChar := -1;
	  RETURN;
	END_IF;
	
	//reset VChar
	#vchar.VelocityLimitPositive := #measuredValues.forward.maxVelocity;
	#vchar.ZeroZonePositive := #measuredValues.forward.minQOutput;
	#vchar.VelocityLimitNegative := #measuredValues.backward.maxVelocity;
	#vchar.ZeroZoneNegative := #measuredValues.backward.minQOutput;
	#vchar.MaxIdx := 0;
	FOR #tempIdx := 0 TO "LSIMAHYD_VCHAR_POINTS_UPPER_LIMIT" DO
	  #vchar.QOutput[#tempIdx] := 0.0;
	  #vchar.Velocity[#tempIdx] := 0.0;
	END_FOR;
	IF #measuredValues.backward.maxIndexMeasurement > 0 THEN
	  FOR #tempIdx := #measuredValues.backward.maxIndexMeasurement TO 1 BY -1 DO
	      #vchar.Velocity[#vchar.MaxIdx] := #measuredValues.backward.velocity[#tempIdx];
	      #vchar.QOutput[#vchar.MaxIdx] := #measuredValues.backward.qOutput[#tempIdx];
	      #vchar.MaxIdx := #vchar.MaxIdx + 1;
	  END_FOR;
	END_IF;
	IF ABS(#vchar.ZeroZoneNegative) > 0.0 THEN
	  #vchar.Velocity[#vchar.MaxIdx] := #measuredValues.backward.velocity[0];
	  #vchar.QOutput[#vchar.MaxIdx] := #measuredValues.backward.qOutput[0];
	  #vchar.MaxIdx := #vchar.MaxIdx + 1;
	END_IF;
	IF #measuredValues.forward.maxIndexMeasurement > 0 THEN
	  FOR #tempIdx := 0 TO #measuredValues.forward.maxIndexMeasurement DO
	    #vchar.Velocity[#vchar.MaxIdx] := #measuredValues.forward.velocity[#tempIdx];
	      #vchar.QOutput[#vchar.MaxIdx] := #measuredValues.forward.qOutput[#tempIdx];
	      #vchar.MaxIdx := #vchar.MaxIdx + 1;
	  END_FOR;
	ELSIF #vchar.ZeroZoneNegative = 0.0 THEN
	  #vchar.Velocity[#vchar.MaxIdx] := #measuredValues.backward.velocity[0];
	  #vchar.QOutput[#vchar.MaxIdx] := #measuredValues.backward.qOutput[0];
	  #vchar.MaxIdx := #vchar.MaxIdx + 1;
	END_IF;
	#vchar.MaxIdx := #vchar.MaxIdx - 1;
	#LSimaHydTO_CreateVChar := 0;
	
	
END_FUNCTION

FUNCTION "SimaHydTO_VCharEditorSortTable" : Void
{ S7_Optimized_Access := 'TRUE' }
FAMILY : SimaHydTO
VERSION : 1.0
   VAR_IN_OUT 
      hmiConnection : "SimaHydTO_typeHMIConnection";
      sortVChar : "LSimaHydTO_typeVCharData";
   END_VAR

   VAR_TEMP 
      tempIndex : Int;
      tempIndex2 : Int;
      tempVCharIndex : Int;
      tempReal : Real;
      tempMinVelocity : Real;
      tempMaxVelocity : Real;
      tempTableLowerBound : DInt;
      tempTableUpperBound : DInt;
   END_VAR

   VAR CONSTANT 
      MAXIMUM_REAL : Real := 0.0;
      MINIMUM_REAL : Real := 0.0;
   END_VAR


BEGIN
	//=============================================================================
	//SIEMENS AG
	//(c)Copyright 2016 All Rights Reserved
	//-----------------------------------------------------------------------------
	//Library:       SimaHydTO_VCharEditorSortTable
	//Tested with:   S7-1500 V2.5
	//Engineering:   TIA Portal V15
	//Restrictions:  -
	//Requirements:  S7-1500(T)
	//Functionality: Sort editor table
	//-----------------------------------------------------------------------------
	//Change log table:
	//Version  Date       Expert in charge Changes applied
	//01.00.00 17.07.2019 ArSc             First released version
	//=============================================================================
	
	"SimaHydTO_GetRealArrayBounds"(lowerBound=>#tempTableLowerBound,
	                               upperBound=>#tempTableUpperBound,
	                               arrayOfReal:=#hmiConnection.VCharEditor.Table.Velocity);
	
	//Save actual table from HMI to VChar data
	FOR #tempIndex := #tempTableLowerBound TO #tempTableUpperBound DO
	  #tempVCharIndex := #tempIndex + #hmiConnection.VCharEditor.Parameter.ActualTableStartIndex;
	  IF ((#tempVCharIndex <= #sortVChar.MaxIdx)
	    AND (#hmiConnection.VCharEditor.Table.Appearance[#tempIndex] > 0))
	  THEN
	    #sortVChar.Velocity[#tempVCharIndex] := #hmiConnection.VCharEditor.Table.Velocity[#tempIndex];
	    #sortVChar.QOutput[#tempVCharIndex] := #hmiConnection.VCharEditor.Table.QOutput[#tempIndex];
	  END_IF;
	END_FOR;
	
	//Reset maximum values
	#tempMinVelocity := #MAXIMUM_REAL;
	#tempMaxVelocity := #MINIMUM_REAL;
	//Sorting
	#tempIndex := 0;
	
	//Sort table  
	REPEAT
	  //Check elements
	  FOR #tempIndex2 := #tempIndex TO #sortVChar.MaxIdx DO
	    //Check minimum and maximum
	    IF (#sortVChar.Velocity[#tempIndex2] > #tempMaxVelocity)
	    THEN
	      #tempMaxVelocity := #sortVChar.Velocity[#tempIndex2];
	    END_IF;
	    IF (#sortVChar.Velocity[#tempIndex2] < #tempMinVelocity)
	    THEN
	      #tempMinVelocity := #sortVChar.Velocity[#tempIndex2];
	    END_IF;
	    //Check for data exchange
	    IF (#sortVChar.QOutput[#tempIndex2] < #sortVChar.QOutput[#tempIndex])
	    THEN
	      //Exchange QOutput
	      #tempReal := #sortVChar.QOutput[#tempIndex];
	      #sortVChar.QOutput[#tempIndex] := #sortVChar.QOutput[#tempIndex2];
	      #sortVChar.QOutput[#tempIndex2] := #tempReal;
	      //Exchange Velocity
	      #tempReal := #sortVChar.Velocity[#tempIndex];
	      #sortVChar.Velocity[#tempIndex] := #sortVChar.Velocity[#tempIndex2];
	      #sortVChar.Velocity[#tempIndex2] := #tempReal;
	    END_IF;
	  END_FOR;
	  //Next line
	  #tempIndex := #tempIndex + 1;
	UNTIL (#tempIndex > #sortVChar.MaxIdx)
	END_REPEAT;
	
	IF #sortVChar.VelocityLimitNegative = 0.0 THEN
	  #sortVChar.VelocityLimitNegative := #tempMinVelocity;
	END_IF;
	IF #sortVChar.VelocityLimitPositive = 0.0 THEN
	  #sortVChar.VelocityLimitPositive := #tempMaxVelocity;
	END_IF;
	
END_FUNCTION

FUNCTION_BLOCK "SimaHydTO_AdvancedAxisControl"
{ S7_Optimized_Access := 'TRUE' }
FAMILY : SimaHydTO
VERSION : 1.0
   VAR_IN_OUT 
      hmiConnection : "SimaHydTO_typeHMIConnection";
      axisData : "LSimaHydTO_typeAxisData";
      axesArray : Array[*] of "SimaHydTO_typeAxesArray";
   END_VAR

   VAR 
      statActualAxisIndex { ExternalAccessible := 'False'; ExternalVisible := 'False'; ExternalWritable := 'False'} : Int;
      statAxisIndexOld { ExternalAccessible := 'False'; ExternalVisible := 'False'; ExternalWritable := 'False'} : Int := -1;
      instSimaHydTO_AxisAdvancedPosAxis { ExternalAccessible := 'False'; ExternalVisible := 'False'; ExternalWritable := 'False'} : "SimaHydTO_AxisAdvanced_PosAxis";
      instSimaHydTO_AxisAdvancedSyncAxis { ExternalAccessible := 'False'; ExternalVisible := 'False'; ExternalWritable := 'False'} : "SimaHydTO_AxisAdvanced_SyncAxis";
   END_VAR


BEGIN
	//=============================================================================
	//SIEMENS AG
	//(c)Copyright 2016 All Rights Reserved
	//-----------------------------------------------------------------------------
	//Library:       SimaHydTO_AdvancedAxisControl
	//Tested with:   S7-1500 V2.5
	//Engineering:   TIA Portal V15
	//Restrictions:  -
	//Requirements:  S7-1500(T)
	//Functionality: Move selected axis
	//-----------------------------------------------------------------------------
	//Change log table:
	//Version  Date       Expert in charge Changes applied
	//01.00.00 19.07.2019 ArSc             First released version
	//=============================================================================
	
	
	//Check axis selection, if axis has changed
	IF #hmiConnection.AxisSelector.Status.selectionChanged
	  AND #hmiConnection.AxisSelector.Status.dataValid
	THEN
	  
	  IF #statAxisIndexOld > -1 THEN  //save axis commands
	    #axesArray[#statAxisIndexOld].advancedControl := #hmiConnection.AdvancedAxisControl.Command;
	  END_IF;
	  
	  
	  //Preset axis commands
	  #statActualAxisIndex := #hmiConnection.AxisSelector.Status.actualAxisIndex;
	  
	  #hmiConnection.AdvancedAxisControl.Command := #axesArray[#statActualAxisIndex].advancedControl;
	  #hmiConnection.AdvancedAxisControl.Command.haltExecute := FALSE;
	  #hmiConnection.AdvancedAxisControl.Command.moveAbsoluteExecute := FALSE;
	  #hmiConnection.AdvancedAxisControl.Command.moveRelativeExecute := FALSE;
	  #statAxisIndexOld := #statActualAxisIndex;
	END_IF;
	
	// workaround for missing dynamics
	#hmiConnection.AdvancedAxisControl.Command.Acceleration := #hmiConnection.BasicAxisControl.Command.jogAcceleration;
	#hmiConnection.AdvancedAxisControl.Command.Deceleration := #hmiConnection.BasicAxisControl.Command.jogDeceleration;
	#hmiConnection.AdvancedAxisControl.Command.Jerk := #hmiConnection.BasicAxisControl.Command.jogJerk;
	
	
	CASE #hmiConnection.AxisSelector.Status.selectedTypeOfAxis OF
	    
	  2: // positioning axis
	    #instSimaHydTO_AxisAdvancedPosAxis(axis := #hmiConnection.AxisSelector.Status.selectedTO_Axis,
	                                       moveRelativeExecute := #hmiConnection.AdvancedAxisControl.Command.moveRelativeExecute,
	                                       moveRelativeDistance := #hmiConnection.AdvancedAxisControl.Command.moveRelativeDistance,
	                                       moveAbsoluteExecute := #hmiConnection.AdvancedAxisControl.Command.moveAbsoluteExecute,
	                                       moveAbsolutePosition := #hmiConnection.AdvancedAxisControl.Command.moveAbsolutePosition,
	                                       moveAbsoluteDirection := #hmiConnection.AdvancedAxisControl.Command.moveAbsoluteDirection,
	                                       haltExecute := #hmiConnection.AdvancedAxisControl.Command.haltExecute,
	                                       haltAbortAcceleration := #hmiConnection.AdvancedAxisControl.Command.haltAbortAcceleration,
	                                       Velocity := #hmiConnection.AdvancedAxisControl.Command.Velocity,
	                                       Acceleration := #hmiConnection.AdvancedAxisControl.Command.Acceleration,
	                                       Deceleration := #hmiConnection.AdvancedAxisControl.Command.Deceleration,
	                                       Jerk := #hmiConnection.AdvancedAxisControl.Command.Jerk,
	                                       moveRelativeDone => #hmiConnection.AdvancedAxisControl.Status.moveRelativeDone,
	                                       moveRelativeBusy => #hmiConnection.AdvancedAxisControl.Status.moveRelativeBusy,
	                                       moveAbsoluteDone => #hmiConnection.AdvancedAxisControl.Status.moveAbsoluteDone,
	                                       moveAbsoluteBusy => #hmiConnection.AdvancedAxisControl.Status.moveAbsoluteBusy,
	                                       haltDone => #hmiConnection.AdvancedAxisControl.Status.haltDone,
	                                       haltBusy => #hmiConnection.AdvancedAxisControl.Status.haltBusy,
	                                       commandAborted => #hmiConnection.AdvancedAxisControl.Status.commandAborted,
	                                       error => #hmiConnection.AdvancedAxisControl.Status.error,
	                                       errorID => #hmiConnection.AdvancedAxisControl.Status.errorID,
	                                       statusID => #hmiConnection.AdvancedAxisControl.Status.statusID);
	    
	    
	  3: // sync axis
	    #instSimaHydTO_AxisAdvancedSyncAxis(axis := #hmiConnection.AxisSelector.Status.selectedTO_Axis,
	                                        moveRelativeExecute := #hmiConnection.AdvancedAxisControl.Command.moveRelativeExecute,
	                                        moveRelativeDistance := #hmiConnection.AdvancedAxisControl.Command.moveRelativeDistance,
	                                        moveAbsoluteExecute := #hmiConnection.AdvancedAxisControl.Command.moveAbsoluteExecute,
	                                        moveAbsolutePosition := #hmiConnection.AdvancedAxisControl.Command.moveAbsolutePosition,
	                                        moveAbsoluteDirection := #hmiConnection.AdvancedAxisControl.Command.moveAbsoluteDirection,
	                                        haltExecute := #hmiConnection.AdvancedAxisControl.Command.haltExecute,
	                                        haltAbortAcceleration := #hmiConnection.AdvancedAxisControl.Command.haltAbortAcceleration,
	                                        Velocity := #hmiConnection.AdvancedAxisControl.Command.Velocity,
	                                        Acceleration := #hmiConnection.AdvancedAxisControl.Command.Acceleration,
	                                        Deceleration := #hmiConnection.AdvancedAxisControl.Command.Deceleration,
	                                        Jerk := #hmiConnection.AdvancedAxisControl.Command.Jerk,
	                                        moveRelativeDone => #hmiConnection.AdvancedAxisControl.Status.moveRelativeDone,
	                                        moveRelativeBusy => #hmiConnection.AdvancedAxisControl.Status.moveRelativeBusy,
	                                        moveAbsoluteDone => #hmiConnection.AdvancedAxisControl.Status.moveAbsoluteDone,
	                                        moveAbsoluteBusy => #hmiConnection.AdvancedAxisControl.Status.moveAbsoluteBusy,
	                                        haltDone => #hmiConnection.AdvancedAxisControl.Status.haltDone,
	                                        haltBusy => #hmiConnection.AdvancedAxisControl.Status.haltBusy,
	                                        commandAborted => #hmiConnection.AdvancedAxisControl.Status.commandAborted,
	                                        error => #hmiConnection.AdvancedAxisControl.Status.error,
	                                        errorID => #hmiConnection.AdvancedAxisControl.Status.errorID,
	                                        statusID => #hmiConnection.AdvancedAxisControl.Status.statusID);
	    
	    
	  ELSE
	    ; // not suported
	    
	END_CASE;
	
END_FUNCTION_BLOCK

